LIN {X 0,Y 368.317,Z 1145.734,A -85,B 0,C 180,E1 7410.615,E2 7410.615} C_VEL
LIN {X 0,Y 379.738,Z 1127.366,A -85,B 0,C 180,E1 7408.419,E2 7408.419} C_VEL
LIN {X 0,Y 392.747,Z 1104.648,A -85,B 0,C 180,E1 7406.175,E2 7406.175} C_VEL
LIN {X 0,Y 402.957,Z 1085.189,A -85,B 0,C 180,E1 7404.57,E2 7404.57} C_VEL
LIN {X 0,Y 412.037,Z 1066.456,A -85,B 0,C 180,E1 7403.257,E2 7403.257} C_VEL
LIN {X 0,Y 421.125,Z 1045.858,A -85,B 0,C 180,E1 7402.016,E2 7402.016} C_VEL
LIN {X 0,Y 431.363,Z 1019.668,A -85,B 0,C 180,E1 7400.719,E2 7400.719} C_VEL
LIN {X 0,Y 438.943,Z 997.212,A -85,B 0,C 180,E1 7399.812,E2 7399.812} C_VEL
LIN {X 0,Y 444.979,Z 976.797,A -85,B 0,C 180,E1 7399.128,E2 7399.128} C_VEL
LIN {X 0,Y 450.336,Z 955.699,A -85,B 0,C 180,E1 7398.541,E2 7398.541} C_VEL
LIN {X 0,Y 455.391,Z 931.712,A -85,B 0,C 180,E1 7398.007,E2 7398.007} C_VEL
LIN {X 0,Y 459.835,Z 902.521,A -85,B 0,C 180,E1 7397.489,E2 7397.489} C_VEL
LIN {X 0,Y 466.482,Z 832.802,A -85,B 0,C 180,E1 7396.426,E2 7396.426} C_VEL
LIN {X 0,Y 482.162,Z 665.13,A -85,B 0,C 180,E1 7393.919,E2 7393.919} C_VEL
LIN {X 0,Y 478.75,Z 659.044,A -85,B 0,C 180,E1 7391.75,E2 7391.75} C_VEL
LIN {X 0,Y 476.474,Z 654.994,A -85,B 0,C 180,E1 7390.031,E2 7390.031} C_VEL
LIN {X 0,Y 474.855,Z 652.158,A -85,B 0,C 180,E1 7388.598,E2 7388.598} C_VEL
LIN {X 0,Y 472.633,Z 648.091,A -85,B 0,C 180,E1 7386.072,E2 7386.072} C_VEL
LIN {X 0,Y 470.733,Z 644.319,A -85,B 0,C 180,E1 7382.191,E2 7382.191} C_VEL
LIN {X 0,Y 470.599,Z 643.362,A -85,B 0,C 180,E1 7381.217,E2 7381.217} C_VEL
LIN {X 0,Y 470.644,Z 643.488,A -85,B 0,C 180,E1 7378.296,E2 7378.296} C_VEL
LIN {X 0,Y 472.388,Z 647.837,A -85,B 0,C 180,E1 7374.047,E2 7374.047} C_VEL
LIN {X 0,Y 473.08,Z 648.922,A -85,B 0,C 180,E1 7373.141,E2 7373.141} C_VEL
LIN {X 0,Y 475.759,Z 653.672,A -85,B 0,C 180,E1 7370.382,E2 7370.382} C_VEL
LIN {X 0,Y 478.483,Z 658.51,A -85,B 0,C 180,E1 7368.244,E2 7368.244} C_VEL
LIN {X 0,Y 481.951,Z 664.628,A -85,B 0,C 180,E1 7366.013,E2 7366.013} C_VEL
LIN {X 0,Y 482.096,Z 665.255,A -85,B 0,C 180,E1 7365.906,E2 7365.906} C_VEL
LIN {X 0,Y 461.587,Z 885.46,A -85,B 0,C 180,E1 7362.619,E2 7362.619} C_VEL
LIN {X 0,Y 458.167,Z 912.997,A -85,B 0,C 180,E1 7362.164,E2 7362.164} C_VEL
LIN {X 0,Y 454.312,Z 935.058,A -85,B 0,C 180,E1 7361.738,E2 7361.738} C_VEL
LIN {X 0,Y 449.575,Z 956.787,A -85,B 0,C 180,E1 7361.215,E2 7361.215} C_VEL
LIN {X 0,Y 442.785,Z 982.701,A -85,B 0,C 180,E1 7360.432,E2 7360.432} C_VEL
LIN {X 0,Y 434.59,Z 1008.147,A -85,B 0,C 180,E1 7359.461,E2 7359.461} C_VEL
LIN {X 0,Y 427.121,Z 1028.517,A -85,B 0,C 180,E1 7358.524,E2 7358.524} C_VEL
LIN {X 0,Y 418.998,Z 1048.357,A -85,B 0,C 180,E1 7357.451,E2 7357.451} C_VEL
LIN {X 0,Y 409.164,Z 1070.092,A -85,B 0,C 180,E1 7356.062,E2 7356.062} C_VEL
LIN {X 0,Y 397.169,Z 1093.722,A -85,B 0,C 180,E1 7354.235,E2 7354.235} C_VEL
LIN {X 0,Y 387.044,Z 1111.972,A -85,B 0,C 180,E1 7352.552,E2 7352.552} C_VEL
LIN {X 0,Y 377.466,Z 1128.083,A -85,B 0,C 180,E1 7350.83,E2 7350.83} C_VEL
LIN {X 0,Y 367.103,Z 1144.491,A -85,B 0,C 180,E1 7348.791,E2 7348.791} C_VEL
LIN {X 0,Y 354.544,Z 1163.366,A -85,B 0,C 180,E1 7346.015,E2 7346.015} C_VEL
LIN {X 0,Y 342.233,Z 1180.606,A -85,B 0,C 180,E1 7342.907,E2 7342.907} C_VEL
LIN {X 0,Y 332.469,Z 1193.855,A -85,B 0,C 180,E1 7340.081,E2 7340.081} C_VEL
LIN {X 0,Y 323.49,Z 1205.781,A -85,B 0,C 180,E1 7337.105,E2 7337.105} C_VEL
LIN {X 0,Y 314.469,Z 1217.64,A -85,B 0,C 180,E1 7333.633,E2 7333.633} C_VEL
LIN {X 0,Y 304.257,Z 1231.131,A -85,B 0,C 180,E1 7328.843,E2 7328.843} C_VEL
LIN {X 0,Y 296.916,Z 1241.098,A -85,B 0,C 180,E1 7324.459,E2 7324.459} C_VEL
LIN {X 0,Y 291.438,Z 1249.004,A -85,B 0,C 180,E1 7320.292,E2 7320.292} C_VEL
LIN {X 0,Y 286.992,Z 1256.043,A -85,B 0,C 180,E1 7315.822,E2 7315.822} C_VEL
LIN {X 0,Y 283.199,Z 1263.061,A -85,B 0,C 180,E1 7310.249,E2 7310.249} C_VEL
LIN {X 0,Y 281.158,Z 1267.846,A -85,B 0,C 180,E1 7305.052,E2 7305.052} C_VEL
LIN {X 0,Y 280.319,Z 1270.683,A -85,B 0,C 180,E1 7300.903,E2 7300.903} C_VEL
LIN {X 0,Y 280.001,Z 1272.679,A -85,B 0,C 180,E1 7296.567,E2 7296.567} C_VEL
LIN {X 0,Y 279.918,Z 1273.647,A -85,B 0,C 180,E1 7292.667,E2 7292.667} C_VEL
LIN {X 0,Y 279.893,Z 1273.817,A -85,B 0,C 180,E1 7288.778,E2 7288.778} C_VEL
LIN {X 0,Y 279.952,Z 1273.12,A -85,B 0,C 180,E1 7284.678,E2 7284.678} C_VEL
LIN {X 0,Y 280.164,Z 1271.42,A -85,B 0,C 180,E1 7280.35,E2 7280.35} C_VEL
LIN {X 0,Y 280.87,Z 1268.724,A -85,B 0,C 180,E1 7275.998,E2 7275.998} C_VEL
LIN {X 0,Y 282.28,Z 1265.011,A -85,B 0,C 180,E1 7271.631,E2 7271.631} C_VEL
LIN {X 0,Y 284.588,Z 1260.252,A -85,B 0,C 180,E1 7267.272,E2 7267.272} C_VEL
LIN {X 0,Y 287.983,Z 1254.413,A -85,B 0,C 180,E1 7262.953,E2 7262.953} C_VEL
LIN {X 0,Y 293.535,Z 1246.053,A -85,B 0,C 180,E1 7257.909,E2 7257.909} C_VEL
LIN {X 0,Y 301.122,Z 1235.389,A -85,B 0,C 180,E1 7252.828,E2 7252.828} C_VEL
LIN {X 0,Y 308.625,Z 1225.359,A -85,B 0,C 180,E1 7248.886,E2 7248.886} C_VEL
LIN {X 0,Y 316.874,Z 1214.522,A -85,B 0,C 180,E1 7245.288,E2 7245.288} C_VEL
LIN {X 0,Y 327.702,Z 1200.432,A -85,B 0,C 180,E1 7241.368,E2 7241.368} C_VEL
LIN {X 0,Y 339.429,Z 1184.587,A -85,B 0,C 180,E1 7237.787,E2 7237.787} C_VEL
LIN {X 0,Y 349.631,Z 1170.387,A -85,B 0,C 180,E1 7235.088,E2 7235.088} C_VEL
LIN {X 0,Y 359.883,Z 1155.548,A -85,B 0,C 180,E1 7232.677,E2 7232.677} C_VEL
LIN {X 0,Y 371.153,Z 1138.435,A -85,B 0,C 180,E1 7230.31,E2 7230.31} C_VEL
LIN {X 0,Y 384.378,Z 1116.814,A -85,B 0,C 180,E1 7227.831,E2 7227.831} C_VEL
LIN {X 0,Y 394.621,Z 1098.654,A -85,B 0,C 180,E1 7226.089,E2 7226.089} C_VEL
LIN {X 0,Y 404.103,Z 1080.565,A -85,B 0,C 180,E1 7224.604,E2 7224.604} C_VEL
LIN {X 0,Y 412.057,Z 1064.18,A -85,B 0,C 180,E1 7223.441,E2 7223.441} C_VEL
LIN {X 0,Y 414.616,Z 1057.936,A -85,B 0,C 180,E1 7222.906,E2 7222.906} C_VEL
LIN {X 0,Y 419.105,Z 1042.697,A -85,B 0,C 180,E1 7221.208,E2 7221.208} C_VEL
LIN {X 0,Y 421.394,Z 1036.166,A -85,B 0,C 180,E1 7220.733,E2 7220.733} C_VEL
LIN {X 0,Y 430.003,Z 1013.794,A -85,B 0,C 180,E1 7219.672,E2 7219.672} C_VEL
LIN {X 0,Y 436.87,Z 993.636,A -85,B 0,C 180,E1 7218.864,E2 7218.864} C_VEL
LIN {X 0,Y 443.002,Z 973.077,A -85,B 0,C 180,E1 7218.173,E2 7218.173} C_VEL
LIN {X 0,Y 448.601,Z 951.126,A -85,B 0,C 180,E1 7217.565,E2 7217.565} C_VEL
LIN {X 0,Y 454.241,Z 923.875,A -85,B 0,C 180,E1 7216.969,E2 7216.969} C_VEL
LIN {X 0,Y 458.06,Z 897.621,A -85,B 0,C 180,E1 7216.52,E2 7216.52} C_VEL
LIN {X 0,Y 474.049,Z 730.963,A -85,B 0,C 180,E1 7214.035,E2 7214.035} C_VEL
LIN {X 0,Y 479.819,Z 670.911,A -85,B 0,C 180,E1 7213.129,E2 7213.129} C_VEL
LIN {X 0,Y 476.073,Z 663.972,A -85,B 0,C 180,E1 7210.467,E2 7210.467} C_VEL
LIN {X 0,Y 473.843,Z 660.068,A -85,B 0,C 180,E1 7208.494,E2 7208.494} C_VEL
LIN {X 0,Y 471.708,Z 656.065,A -85,B 0,C 180,E1 7205.962,E2 7205.962} C_VEL
LIN {X 0,Y 469.919,Z 652.326,A -85,B 0,C 180,E1 7201.951,E2 7201.951} C_VEL
LIN {X 0,Y 469.825,Z 651.372,A -85,B 0,C 180,E1 7200.854,E2 7200.854} C_VEL
LIN {X 0,Y 469.866,Z 651.609,A -85,B 0,C 180,E1 7198.781,E2 7198.781} C_VEL
LIN {X 0,Y 471.112,Z 655.393,A -85,B 0,C 180,E1 7195.008,E2 7195.008} C_VEL
LIN {X 0,Y 472.091,Z 656.797,A -85,B 0,C 180,E1 7193.616,E2 7193.616} C_VEL
LIN {X 0,Y 474.785,Z 661.714,A -85,B 0,C 180,E1 7190.729,E2 7190.729} C_VEL
LIN {X 0,Y 477.278,Z 666.333,A -85,B 0,C 180,E1 7188.704,E2 7188.704} C_VEL
LIN {X 0,Y 479.903,Z 671.155,A -85,B 0,C 180,E1 7186.921,E2 7186.921} C_VEL
LIN {X 0,Y 459.204,Z 888.928,A -85,B 0,C 180,E1 7183.693,E2 7183.693} C_VEL
LIN {X 0,Y 455.746,Z 916.161,A -85,B 0,C 180,E1 7183.247,E2 7183.247} C_VEL
LIN {X 0,Y 451.785,Z 938.355,A -85,B 0,C 180,E1 7182.831,E2 7182.831} C_VEL
LIN {X 0,Y 446.979,Z 959.904,A -85,B 0,C 180,E1 7182.335,E2 7182.335} C_VEL
LIN {X 0,Y 440.355,Z 984.664,A -85,B 0,C 180,E1 7181.626,E2 7181.626} C_VEL
LIN {X 0,Y 431.937,Z 1010.547,A -85,B 0,C 180,E1 7180.684,E2 7180.684} C_VEL
LIN {X 0,Y 424.106,Z 1031.526,A -85,B 0,C 180,E1 7179.756,E2 7179.756} C_VEL
LIN {X 0,Y 416.174,Z 1050.594,A -85,B 0,C 180,E1 7178.762,E2 7178.762} C_VEL
LIN {X 0,Y 407.238,Z 1070.13,A -85,B 0,C 180,E1 7177.563,E2 7177.563} C_VEL
LIN {X 0,Y 395.845,Z 1092.788,A -85,B 0,C 180,E1 7175.926,E2 7175.926} C_VEL
LIN {X 0,Y 383.686,Z 1114.369,A -85,B 0,C 180,E1 7174.021,E2 7174.021} C_VEL
LIN {X 0,Y 373.027,Z 1131.965,A -85,B 0,C 180,E1 7172.182,E2 7172.182} C_VEL
LIN {X 0,Y 362.443,Z 1148.392,A -85,B 0,C 180,E1 7170.17,E2 7170.17} C_VEL
LIN {X 0,Y 349.788,Z 1166.999,A -85,B 0,C 180,E1 7167.475,E2 7167.475} C_VEL
LIN {X 0,Y 337.022,Z 1184.513,A -85,B 0,C 180,E1 7164.369,E2 7164.369} C_VEL
LIN {X 0,Y 326.887,Z 1197.959,A -85,B 0,C 180,E1 7161.53,E2 7161.53} C_VEL
LIN {X 0,Y 317.538,Z 1210.075,A -85,B 0,C 180,E1 7158.53,E2 7158.53} C_VEL
LIN {X 0,Y 308.117,Z 1222.135,A -85,B 0,C 180,E1 7155.017,E2 7155.017} C_VEL
LIN {X 0,Y 297.906,Z 1235.366,A -85,B 0,C 180,E1 7150.365,E2 7150.365} C_VEL
LIN {X 0,Y 289.742,Z 1246.09,A -85,B 0,C 180,E1 7145.668,E2 7145.668} C_VEL
LIN {X 0,Y 283.977,Z 1254.183,A -85,B 0,C 180,E1 7141.398,E2 7141.398} C_VEL
LIN {X 0,Y 279.444,Z 1261.114,A -85,B 0,C 180,E1 7137.006,E2 7137.006} C_VEL
LIN {X 0,Y 275.889,Z 1267.394,A -85,B 0,C 180,E1 7132.136,E2 7132.136} C_VEL
LIN {X 0,Y 273.308,Z 1273.104,A -85,B 0,C 180,E1 7126.355,E2 7126.355} C_VEL
LIN {X 0,Y 272.278,Z 1276.597,A -85,B 0,C 180,E1 7121.33,E2 7121.33} C_VEL
LIN {X 0,Y 271.97,Z 1278.637,A -85,B 0,C 180,E1 7116.949,E2 7116.949} C_VEL
LIN {X 0,Y 271.913,Z 1279.663,A -85,B 0,C 180,E1 7112.945,E2 7112.945} C_VEL
LIN {X 0,Y 271.897,Z 1279.844,A -85,B 0,C 180,E1 7108.73,E2 7108.73} C_VEL
LIN {X 0,Y 271.931,Z 1279.107,A -85,B 0,C 180,E1 7104.508,E2 7104.508} C_VEL
LIN {X 0,Y 272.089,Z 1277.448,A -85,B 0,C 180,E1 7100.262,E2 7100.262} C_VEL
LIN {X 0,Y 272.771,Z 1274.701,A -85,B 0,C 180,E1 7095.777,E2 7095.777} C_VEL
LIN {X 0,Y 274.181,Z 1270.916,A -85,B 0,C 180,E1 7091.276,E2 7091.276} C_VEL
LIN {X 0,Y 276.532,Z 1266.069,A -85,B 0,C 180,E1 7086.783,E2 7086.783} C_VEL
LIN {X 0,Y 279.837,Z 1260.434,A -85,B 0,C 180,E1 7082.548,E2 7082.548} C_VEL
LIN {X 0,Y 284.734,Z 1253.054,A -85,B 0,C 180,E1 7077.972,E2 7077.972} C_VEL
LIN {X 0,Y 292.301,Z 1242.694,A -85,B 0,C 180,E1 7072.732,E2 7072.732} C_VEL
LIN {X 0,Y 301.068,Z 1231.11,A -85,B 0,C 180,E1 7068.068,E2 7068.068} C_VEL
LIN {X 0,Y 309.48,Z 1220.307,A -85,B 0,C 180,E1 7064.432,E2 7064.432} C_VEL
LIN {X 0,Y 319.243,Z 1207.822,A -85,B 0,C 180,E1 7060.89,E2 7060.89} C_VEL
LIN {X 0,Y 331.907,Z 1191.336,A -85,B 0,C 180,E1 7057.025,E2 7057.025} C_VEL
LIN {X 0,Y 343.634,Z 1175.359,A -85,B 0,C 180,E1 7053.964,E2 7053.964} C_VEL
LIN {X 0,Y 353.856,Z 1160.909,A -85,B 0,C 180,E1 7051.618,E2 7051.618} C_VEL
LIN {X 0,Y 364.151,Z 1145.639,A -85,B 0,C 180,E1 7049.488,E2 7049.488} C_VEL
LIN {X 0,Y 375.653,Z 1127.607,A -85,B 0,C 180,E1 7047.345,E2 7047.345} C_VEL
LIN {X 0,Y 389.207,Z 1104.505,A -85,B 0,C 180,E1 7045.081,E2 7045.081} C_VEL
LIN {X 0,Y 399.609,Z 1085.094,A -85,B 0,C 180,E1 7043.498,E2 7043.498} C_VEL
LIN {X 0,Y 408.802,Z 1066.504,A -85,B 0,C 180,E1 7042.211,E2 7042.211} C_VEL
LIN {X 0,Y 417.778,Z 1046.575,A -85,B 0,C 180,E1 7041.024,E2 7041.024} C_VEL
LIN {X 0,Y 428.155,Z 1020.705,A -85,B 0,C 180,E1 7039.752,E2 7039.752} C_VEL
LIN {X 0,Y 436.117,Z 997.583,A -85,B 0,C 180,E1 7038.828,E2 7038.828} C_VEL
LIN {X 0,Y 442.334,Z 976.931,A -85,B 0,C 180,E1 7038.147,E2 7038.147} C_VEL
LIN {X 0,Y 447.76,Z 955.926,A -85,B 0,C 180,E1 7037.572,E2 7037.572} C_VEL
LIN {X 0,Y 452.756,Z 932.675,A -85,B 0,C 180,E1 7037.061,E2 7037.061} C_VEL
LIN {X 0,Y 457.442,Z 902.766,A -85,B 0,C 180,E1 7036.534,E2 7036.534} C_VEL
LIN {X 0,Y 463.818,Z 837.541,A -85,B 0,C 180,E1 7035.546,E2 7035.546} C_VEL
LIN {X 0,Y 479.71,Z 670.904,A -85,B 0,C 180,E1 7033.071,E2 7033.071} C_VEL
LIN {X 0,Y 475.936,Z 663.895,A -85,B 0,C 180,E1 7030.409,E2 7030.409} C_VEL
LIN {X 0,Y 473.747,Z 660.045,A -85,B 0,C 180,E1 7028.496,E2 7028.496} C_VEL
LIN {X 0,Y 471.564,Z 655.972,A -85,B 0,C 180,E1 7025.964,E2 7025.964} C_VEL
LIN {X 0,Y 469.727,Z 652.2,A -85,B 0,C 180,E1 7022.074,E2 7022.074} C_VEL
LIN {X 0,Y 469.602,Z 651.303,A -85,B 0,C 180,E1 7021.098,E2 7021.098} C_VEL
LIN {X 0,Y 469.657,Z 651.529,A -85,B 0,C 180,E1 7018.292,E2 7018.292} C_VEL
LIN {X 0,Y 471.506,Z 655.906,A -85,B 0,C 180,E1 7013.913,E2 7013.913} C_VEL
LIN {X 0,Y 474.501,Z 661.361,A -85,B 0,C 180,E1 7010.601,E2 7010.601} C_VEL
LIN {X 0,Y 477.157,Z 666.206,A -85,B 0,C 180,E1 7008.456,E2 7008.456} C_VEL
LIN {X 0,Y 479.675,Z 670.8,A -85,B 0,C 180,E1 7006.755,E2 7006.755} C_VEL
LIN {X 0,Y 458.737,Z 890.156,A -85,B 0,C 180,E1 7003.501,E2 7003.501} C_VEL
LIN {X 0,Y 455.594,Z 914.237,A -85,B 0,C 180,E1 7003.104,E2 7003.104} C_VEL
LIN {X 0,Y 451.679,Z 936.071,A -85,B 0,C 180,E1 7002.685,E2 7002.685} C_VEL
LIN {X 0,Y 446.64,Z 958.608,A -85,B 0,C 180,E1 7002.146,E2 7002.146} C_VEL
LIN {X 0,Y 438.862,Z 986.854,A -85,B 0,C 180,E1 7001.281,E2 7001.281} C_VEL
LIN {X 0,Y 431.414,Z 1009.371,A -85,B 0,C 180,E1 7000.419,E2 7000.419} C_VEL
LIN {X 0,Y 423.82,Z 1029.615,A -85,B 0,C 180,E1 6999.494,E2 6999.494} C_VEL
LIN {X 0,Y 415.522,Z 1049.426,A -85,B 0,C 180,E1 6998.431,E2 6998.431} C_VEL
LIN {X 0,Y 404.396,Z 1073.352,A -85,B 0,C 180,E1 6996.899,E2 6996.899} C_VEL
LIN {X 0,Y 393.143,Z 1094.765,A -85,B 0,C 180,E1 6995.23,E2 6995.23} C_VEL
LIN {X 0,Y 383.352,Z 1112.005,A -85,B 0,C 180,E1 6993.651,E2 6993.651} C_VEL
LIN {X 0,Y 373.422,Z 1128.307,A -85,B 0,C 180,E1 6991.923,E2 6991.923} C_VEL
LIN {X 0,Y 362.775,Z 1144.736,A -85,B 0,C 180,E1 6989.892,E2 6989.892} C_VEL
LIN {X 0,Y 349.751,Z 1163.743,A -85,B 0,C 180,E1 6987.099,E2 6987.099} C_VEL
LIN {X 0,Y 337.257,Z 1180.7,A -85,B 0,C 180,E1 6984.04,E2 6984.04} C_VEL
LIN {X 0,Y 327.152,Z 1193.959,A -85,B 0,C 180,E1 6981.204,E2 6981.204} C_VEL
LIN {X 0,Y 317.349,Z 1206.506,A -85,B 0,C 180,E1 6978.042,E2 6978.042} C_VEL
LIN {X 0,Y 306.719,Z 1220.011,A -85,B 0,C 180,E1 6973.982,E2 6973.982} C_VEL
LIN {X 0,Y 296.734,Z 1232.51,A -85,B 0,C 180,E1 6969.313,E2 6969.313} C_VEL
LIN {X 0,Y 289.758,Z 1241.592,A -85,B 0,C 180,E1 6965.194,E2 6965.194} C_VEL
LIN {X 0,Y 284.027,Z 1249.446,A -85,B 0,C 180,E1 6960.934,E2 6960.934} C_VEL
LIN {X 0,Y 278.966,Z 1257.098,A -85,B 0,C 180,E1 6955.887,E2 6955.887} C_VEL
LIN {X 0,Y 275.042,Z 1263.966,A -85,B 0,C 180,E1 6949.988,E2 6949.988} C_VEL
LIN {X 0,Y 273.214,Z 1268.093,A -85,B 0,C 180,E1 6945.283,E2 6945.283} C_VEL
LIN {X 0,Y 272.335,Z 1270.884,A -85,B 0,C 180,E1 6941.012,E2 6941.012} C_VEL
LIN {X 0,Y 272.008,Z 1272.767,A -85,B 0,C 180,E1 6936.761,E2 6936.761} C_VEL
LIN {X 0,Y 271.919,Z 1273.735,A -85,B 0,C 180,E1 6932.746,E2 6932.746} C_VEL
LIN {X 0,Y 271.896,Z 1273.904,A -85,B 0,C 180,E1 6928.742,E2 6928.742} C_VEL
LIN {X 0,Y 271.957,Z 1273.208,A -85,B 0,C 180,E1 6924.521,E2 6924.521} C_VEL
LIN {X 0,Y 272.186,Z 1271.508,A -85,B 0,C 180,E1 6920.064,E2 6920.064} C_VEL
LIN {X 0,Y 272.968,Z 1268.813,A -85,B 0,C 180,E1 6915.584,E2 6915.584} C_VEL
LIN {X 0,Y 274.49,Z 1265.1,A -85,B 0,C 180,E1 6911.09,E2 6911.09} C_VEL
LIN {X 0,Y 276.97,Z 1260.341,A -85,B 0,C 180,E1 6906.61,E2 6906.61} C_VEL
LIN {X 0,Y 280.597,Z 1254.503,A -85,B 0,C 180,E1 6902.181,E2 6902.181} C_VEL
LIN {X 0,Y 286.485,Z 1246.143,A -85,B 0,C 180,E1 6897.02,E2 6897.02} C_VEL
LIN {X 0,Y 294.492,Z 1235.479,A -85,B 0,C 180,E1 6891.843,E2 6891.843} C_VEL
LIN {X 0,Y 302.347,Z 1225.449,A -85,B 0,C 180,E1 6887.839,E2 6887.839} C_VEL
LIN {X 0,Y 310.97,Z 1214.612,A -85,B 0,C 180,E1 6884.2,E2 6884.2} C_VEL
LIN {X 0,Y 322.229,Z 1200.522,A -85,B 0,C 180,E1 6880.251,E2 6880.251} C_VEL
LIN {X 0,Y 334.193,Z 1184.921,A -85,B 0,C 180,E1 6876.706,E2 6876.706} C_VEL
LIN {X 0,Y 344.807,Z 1170.617,A -85,B 0,C 180,E1 6873.98,E2 6873.98} C_VEL
LIN {X 0,Y 355.468,Z 1155.636,A -85,B 0,C 180,E1 6871.55,E2 6871.55} C_VEL
LIN {X 0,Y 367.136,Z 1138.387,A -85,B 0,C 180,E1 6869.177,E2 6869.177} C_VEL
LIN {X 0,Y 380.601,Z 1116.9,A -85,B 0,C 180,E1 6866.734,E2 6866.734} C_VEL
LIN {X 0,Y 391.078,Z 1098.74,A -85,B 0,C 180,E1 6865.008,E2 6865.008} C_VEL
LIN {X 0,Y 400.88,Z 1080.414,A -85,B 0,C 180,E1 6863.521,E2 6863.521} C_VEL
LIN {X 0,Y 409.928,Z 1062.06,A -85,B 0,C 180,E1 6862.248,E2 6862.248} C_VEL
LIN {X 0,Y 420.216,Z 1039.054,A -85,B 0,C 180,E1 6860.884,E2 6860.884} C_VEL
LIN {X 0,Y 421.394,Z 1036.166,A -85,B 0,C 180,E1 6860.733,E2 6860.733} C_VEL
LIN {X 0,Y 423.713,Z 1029.54,A -85,B 0,C 180,E1 6860.279,E2 6860.279} C_VEL
LIN {X 0,Y 428.122,Z 1012.463,A -85,B 0,C 180,E1 6858.69,E2 6858.69} C_VEL
LIN {X 0,Y 429.972,Z 1006.631,A -85,B 0,C 180,E1 6858.346,E2 6858.346} C_VEL
LIN {X 0,Y 438.893,Z 979.066,A -85,B 0,C 180,E1 6857.359,E2 6857.359} C_VEL
LIN {X 0,Y 445.082,Z 955.962,A -85,B 0,C 180,E1 6856.699,E2 6856.699} C_VEL
LIN {X 0,Y 449.846,Z 934.642,A -85,B 0,C 180,E1 6856.209,E2 6856.209} C_VEL
LIN {X 0,Y 453.871,Z 912.105,A -85,B 0,C 180,E1 6855.79,E2 6855.79} C_VEL
LIN {X 0,Y 457.572,Z 882.153,A -85,B 0,C 180,E1 6855.312,E2 6855.312} C_VEL
LIN {X 0,Y 477.509,Z 676.816,A -85,B 0,C 180,E1 6852.294,E2 6852.294} C_VEL
LIN {X 0,Y 474.281,Z 670.822,A -85,B 0,C 180,E1 6849.832,E2 6849.832} C_VEL
LIN {X 0,Y 472.616,Z 667.782,A -85,B 0,C 180,E1 6848.272,E2 6848.272} C_VEL
LIN {X 0,Y 470.643,Z 663.947,A -85,B 0,C 180,E1 6845.853,E2 6845.853} C_VEL
LIN {X 0,Y 468.92,Z 660.205,A -85,B 0,C 180,E1 6841.833,E2 6841.833} C_VEL
LIN {X 0,Y 468.836,Z 659.318,A -85,B 0,C 180,E1 6840.733,E2 6840.733} C_VEL
LIN {X 0,Y 468.883,Z 659.62,A -85,B 0,C 180,E1 6838.778,E2 6838.778} C_VEL
LIN {X 0,Y 470.135,Z 663.376,A -85,B 0,C 180,E1 6834.997,E2 6834.997} C_VEL
LIN {X 0,Y 471.013,Z 664.714,A -85,B 0,C 180,E1 6833.723,E2 6833.723} C_VEL
LIN {X 0,Y 473.596,Z 669.536,A -85,B 0,C 180,E1 6830.889,E2 6830.889} C_VEL
LIN {X 0,Y 476.04,Z 674.176,A -85,B 0,C 180,E1 6828.858,E2 6828.858} C_VEL
LIN {X 0,Y 477.549,Z 677.122,A -85,B 0,C 180,E1 6827.772,E2 6827.772} C_VEL
LIN {X 0,Y 456.473,Z 893.486,A -85,B 0,C 180,E1 6824.588,E2 6824.588} C_VEL
LIN {X 0,Y 453.312,Z 917.226,A -85,B 0,C 180,E1 6824.199,E2 6824.199} C_VEL
LIN {X 0,Y 449.265,Z 939.323,A -85,B 0,C 180,E1 6823.789,E2 6823.789} C_VEL
LIN {X 0,Y 443.992,Z 962.337,A -85,B 0,C 180,E1 6823.262,E2 6823.262} C_VEL
LIN {X 0,Y 435.92,Z 990.787,A -85,B 0,C 180,E1 6822.424,E2 6822.424} C_VEL
LIN {X 0,Y 428.73,Z 1012.087,A -85,B 0,C 180,E1 6821.64,E2 6821.64} C_VEL
LIN {X 0,Y 421.359,Z 1031.443,A -85,B 0,C 180,E1 6820.794,E2 6820.794} C_VEL
LIN {X 0,Y 413.287,Z 1050.51,A -85,B 0,C 180,E1 6819.817,E2 6819.817} C_VEL
LIN {X 0,Y 404.181,Z 1070.046,A -85,B 0,C 180,E1 6818.637,E2 6818.637} C_VEL
LIN {X 0,Y 392.174,Z 1093.382,A -85,B 0,C 180,E1 6816.968,E2 6816.968} C_VEL
LIN {X 0,Y 380.134,Z 1114.282,A -85,B 0,C 180,E1 6815.142,E2 6815.142} C_VEL
LIN {X 0,Y 369.228,Z 1131.878,A -85,B 0,C 180,E1 6813.321,E2 6813.321} C_VEL
LIN {X 0,Y 358.363,Z 1148.327,A -85,B 0,C 180,E1 6811.321,E2 6811.321} C_VEL
LIN {X 0,Y 345.37,Z 1166.911,A -85,B 0,C 180,E1 6808.642,E2 6808.642} C_VEL
LIN {X 0,Y 332.163,Z 1184.48,A -85,B 0,C 180,E1 6805.533,E2 6805.533} C_VEL
LIN {X 0,Y 321.703,Z 1197.903,A -85,B 0,C 180,E1 6802.693,E2 6802.693} C_VEL
LIN {X 0,Y 311.514,Z 1210.624,A -85,B 0,C 180,E1 6799.516,E2 6799.516} C_VEL
LIN {X 0,Y 300.85,Z 1223.776,A -85,B 0,C 180,E1 6795.597,E2 6795.597} C_VEL
LIN {X 0,Y 289.982,Z 1237.126,A -85,B 0,C 180,E1 6790.659,E2 6790.659} C_VEL
LIN {X 0,Y 282.636,Z 1246.408,A -85,B 0,C 180,E1 6786.456,E2 6786.456} C_VEL
LIN {X 0,Y 276.605,Z 1254.449,A -85,B 0,C 180,E1 6782.09,E2 6782.09} C_VEL
LIN {X 0,Y 271.665,Z 1261.617,A -85,B 0,C 180,E1 6777.384,E2 6777.384} C_VEL
LIN {X 0,Y 267.419,Z 1268.839,A -85,B 0,C 180,E1 6771.405,E2 6771.405} C_VEL
LIN {X 0,Y 265.244,Z 1273.501,A -85,B 0,C 180,E1 6766.191,E2 6766.191} C_VEL
LIN {X 0,Y 264.302,Z 1276.588,A -85,B 0,C 180,E1 6761.525,E2 6761.525} C_VEL
LIN {X 0,Y 263.973,Z 1278.582,A -85,B 0,C 180,E1 6757.058,E2 6757.058} C_VEL
LIN {X 0,Y 263.913,Z 1279.599,A -85,B 0,C 180,E1 6752.817,E2 6752.817} C_VEL
LIN {X 0,Y 263.898,Z 1279.757,A -85,B 0,C 180,E1 6748.691,E2 6748.691} C_VEL
LIN {X 0,Y 263.934,Z 1279.019,A -85,B 0,C 180,E1 6744.341,E2 6744.341} C_VEL
LIN {X 0,Y 264.121,Z 1277.289,A -85,B 0,C 180,E1 6739.832,E2 6739.832} C_VEL
LIN {X 0,Y 264.864,Z 1274.611,A -85,B 0,C 180,E1 6735.343,E2 6735.343} C_VEL
LIN {X 0,Y 266.397,Z 1270.825,A -85,B 0,C 180,E1 6730.708,E2 6730.708} C_VEL
LIN {X 0,Y 268.928,Z 1265.977,A -85,B 0,C 180,E1 6726.087,E2 6726.087} C_VEL
LIN {X 0,Y 272.462,Z 1260.337,A -85,B 0,C 180,E1 6721.735,E2 6721.735} C_VEL
LIN {X 0,Y 277.394,Z 1253.318,A -85,B 0,C 180,E1 6717.264,E2 6717.264} C_VEL
LIN {X 0,Y 285.315,Z 1243.059,A -85,B 0,C 180,E1 6711.912,E2 6711.912} C_VEL
LIN {X 0,Y 294.372,Z 1231.621,A -85,B 0,C 180,E1 6707.196,E2 6707.196} C_VEL
LIN {X 0,Y 303.176,Z 1220.791,A -85,B 0,C 180,E1 6703.479,E2 6703.479} C_VEL
LIN {X 0,Y 312.571,Z 1209.229,A -85,B 0,C 180,E1 6700.129,E2 6700.129} C_VEL
LIN {X 0,Y 324.028,Z 1194.914,A -85,B 0,C 180,E1 6696.644,E2 6696.644} C_VEL
LIN {X 0,Y 337.765,Z 1176.982,A -85,B 0,C 180,E1 6693.09,E2 6693.09} C_VEL
LIN {X 0,Y 348.965,Z 1161.64,A -85,B 0,C 180,E1 6690.576,E2 6690.576} C_VEL
LIN {X 0,Y 359.438,Z 1146.563,A -85,B 0,C 180,E1 6688.467,E2 6688.467} C_VEL
LIN {X 0,Y 369.97,Z 1130.522,A -85,B 0,C 180,E1 6686.543,E2 6686.543} C_VEL
LIN {X 0,Y 382.391,Z 1110.344,A -85,B 0,C 180,E1 6684.496,E2 6684.496} C_VEL
LIN {X 0,Y 395.249,Z 1087.21,A -85,B 0,C 180,E1 6682.573,E2 6682.573} C_VEL
LIN {X 0,Y 405.086,Z 1067.834,A -85,B 0,C 180,E1 6681.231,E2 6681.231} C_VEL
LIN {X 0,Y 413.715,Z 1049.187,A -85,B 0,C 180,E1 6680.12,E2 6680.12} C_VEL
LIN {X 0,Y 422.204,Z 1028.957,A -85,B 0,C 180,E1 6679.098,E2 6679.098} C_VEL
LIN {X 0,Y 431.657,Z 1003.454,A -85,B 0,C 180,E1 6678.029,E2 6678.029} C_VEL
LIN {X 0,Y 439.257,Z 979.058,A -85,B 0,C 180,E1 6677.213,E2 6677.213} C_VEL
LIN {X 0,Y 444.945,Z 957.673,A -85,B 0,C 180,E1 6676.629,E2 6676.629} C_VEL
LIN {X 0,Y 449.718,Z 936.208,A -85,B 0,C 180,E1 6676.155,E2 6676.155} C_VEL
LIN {X 0,Y 454.156,Z 910.846,A -85,B 0,C 180,E1 6675.697,E2 6675.697} C_VEL
LIN {X 0,Y 458.264,Z 873.736,A -85,B 0,C 180,E1 6675.122,E2 6675.122} C_VEL
LIN {X 0,Y 477.37,Z 676.767,A -85,B 0,C 180,E1 6672.223,E2 6672.223} C_VEL
LIN {X 0,Y 474.135,Z 670.741,A -85,B 0,C 180,E1 6669.774,E2 6669.774} C_VEL
LIN {X 0,Y 472.392,Z 667.581,A -85,B 0,C 180,E1 6668.153,E2 6668.153} C_VEL
LIN {X 0,Y 470.406,Z 663.755,A -85,B 0,C 180,E1 6665.734,E2 6665.734} C_VEL
LIN {X 0,Y 468.707,Z 659.928,A -85,B 0,C 180,E1 6661.834,E2 6661.834} C_VEL
LIN {X 0,Y 468.607,Z 659.246,A -85,B 0,C 180,E1 6660.978,E2 6660.978} C_VEL
LIN {X 0,Y 468.663,Z 659.411,A -85,B 0,C 180,E1 6658.411,E2 6658.411} C_VEL
LIN {X 0,Y 470.44,Z 663.788,A -85,B 0,C 180,E1 6654.022,E2 6654.022} C_VEL
LIN {X 0,Y 473.25,Z 669.051,A -85,B 0,C 180,E1 6650.821,E2 6650.821} C_VEL
LIN {X 0,Y 475.917,Z 674.051,A -85,B 0,C 180,E1 6648.61,E2 6648.61} C_VEL
LIN {X 0,Y 477.315,Z 676.801,A -85,B 0,C 180,E1 6647.606,E2 6647.606} C_VEL
LIN {X 0,Y 456.2,Z 893.047,A -85,B 0,C 180,E1 6644.423,E2 6644.423} C_VEL
LIN {X 0,Y 453.118,Z 915.639,A -85,B 0,C 180,E1 6644.052,E2 6644.052} C_VEL
LIN {X 0,Y 449.039,Z 937.734,A -85,B 0,C 180,E1 6643.63,E2 6643.63} C_VEL
LIN {X 0,Y 443.064,Z 963.621,A -85,B 0,C 180,E1 6643.003,E2 6643.003} C_VEL
LIN {X 0,Y 435.768,Z 988.708,A -85,B 0,C 180,E1 6642.224,E2 6642.224} C_VEL
LIN {X 0,Y 428.769,Z 1009.467,A -85,B 0,C 180,E1 6641.438,E2 6641.438} C_VEL
LIN {X 0,Y 421.046,Z 1029.71,A -85,B 0,C 180,E1 6640.528,E2 6640.528} C_VEL
LIN {X 0,Y 412.631,Z 1049.445,A -85,B 0,C 180,E1 6639.487,E2 6639.487} C_VEL
LIN {X 0,Y 401.261,Z 1073.446,A -85,B 0,C 180,E1 6637.972,E2 6637.972} C_VEL
LIN {X 0,Y 389.543,Z 1095.274,A -85,B 0,C 180,E1 6636.289,E2 6636.289} C_VEL
LIN {X 0,Y 379.633,Z 1112.322,A -85,B 0,C 180,E1 6634.743,E2 6634.743} C_VEL
LIN {X 0,Y 369.248,Z 1128.954,A -85,B 0,C 180,E1 6632.991,E2 6632.991} C_VEL
LIN {X 0,Y 357.769,Z 1146.193,A -85,B 0,C 180,E1 6630.857,E2 6630.857} C_VEL
LIN {X 0,Y 342.943,Z 1166.925,A -85,B 0,C 180,E1 6627.733,E2 6627.733} C_VEL
LIN {X 0,Y 331.821,Z 1181.56,A -85,B 0,C 180,E1 6625.052,E2 6625.052} C_VEL
LIN {X 0,Y 321.424,Z 1194.739,A -85,B 0,C 180,E1 6622.204,E2 6622.204} C_VEL
LIN {X 0,Y 311.298,Z 1207.231,A -85,B 0,C 180,E1 6619.015,E2 6619.015} C_VEL
LIN {X 0,Y 299.846,Z 1221.193,A -85,B 0,C 180,E1 6614.723,E2 6614.723} C_VEL
LIN {X 0,Y 289.918,Z 1233.058,A -85,B 0,C 180,E1 6610.166,E2 6610.166} C_VEL
LIN {X 0,Y 282.967,Z 1241.685,A -85,B 0,C 180,E1 6606.17,E2 6606.17} C_VEL
LIN {X 0,Y 276.91,Z 1249.538,A -85,B 0,C 180,E1 6601.821,E2 6601.821} C_VEL
LIN {X 0,Y 271.565,Z 1257.126,A -85,B 0,C 180,E1 6596.698,E2 6596.698} C_VEL
LIN {X 0,Y 267.313,Z 1264.057,A -85,B 0,C 180,E1 6590.591,E2 6590.591} C_VEL
LIN {X 0,Y 265.334,Z 1268.183,A -85,B 0,C 180,E1 6585.749,E2 6585.749} C_VEL
LIN {X 0,Y 264.392,Z 1270.973,A -85,B 0,C 180,E1 6581.347,E2 6581.347} C_VEL
LIN {X 0,Y 264.018,Z 1272.855,A -85,B 0,C 180,E1 6576.967,E2 6576.967} C_VEL
LIN {X 0,Y 263.92,Z 1273.823,A -85,B 0,C 180,E1 6572.829,E2 6572.829} C_VEL
LIN {X 0,Y 263.897,Z 1273.992,A -85,B 0,C 180,E1 6568.704,E2 6568.704} C_VEL
LIN {X 0,Y 263.963,Z 1273.296,A -85,B 0,C 180,E1 6564.354,E2 6564.354} C_VEL
LIN {X 0,Y 264.196,Z 1271.708,A -85,B 0,C 180,E1 6559.981,E2 6559.981} C_VEL
LIN {X 0,Y 265.02,Z 1269.059,A -85,B 0,C 180,E1 6555.365,E2 6555.365} C_VEL
LIN {X 0,Y 266.625,Z 1265.393,A -85,B 0,C 180,E1 6550.738,E2 6550.738} C_VEL
LIN {X 0,Y 269.24,Z 1260.682,A -85,B 0,C 180,E1 6546.129,E2 6546.129} C_VEL
LIN {X 0,Y 272.846,Z 1255.192,A -85,B 0,C 180,E1 6541.796,E2 6541.796} C_VEL
LIN {X 0,Y 277.85,Z 1248.331,A -85,B 0,C 180,E1 6537.339,E2 6537.339} C_VEL
LIN {X 0,Y 285.137,Z 1239.09,A -85,B 0,C 180,E1 6532.408,E2 6532.408} C_VEL
LIN {X 0,Y 294.933,Z 1227.071,A -85,B 0,C 180,E1 6527.319,E2 6527.319} C_VEL
LIN {X 0,Y 303.76,Z 1216.409,A -85,B 0,C 180,E1 6523.611,E2 6523.611} C_VEL
LIN {X 0,Y 313.168,Z 1205.027,A -85,B 0,C 180,E1 6520.275,E2 6520.275} C_VEL
LIN {X 0,Y 323.83,Z 1191.874,A -85,B 0,C 180,E1 6517.021,E2 6517.021} C_VEL
LIN {X 0,Y 338.344,Z 1173.228,A -85,B 0,C 180,E1 6513.258,E2 6513.258} C_VEL
LIN {X 0,Y 349.538,Z 1158.028,A -85,B 0,C 180,E1 6510.741,E2 6510.741} C_VEL
LIN {X 0,Y 360.298,Z 1142.647,A -85,B 0,C 180,E1 6508.572,E2 6508.572} C_VEL
LIN {X 0,Y 371.173,Z 1126.171,A -85,B 0,C 180,E1 6506.589,E2 6506.589} C_VEL
LIN {X 0,Y 384.322,Z 1104.814,A -85,B 0,C 180,E1 6504.429,E2 6504.429} C_VEL
LIN {X 0,Y 396.408,Z 1082.932,A -85,B 0,C 180,E1 6502.621,E2 6502.621} C_VEL
LIN {X 0,Y 405.73,Z 1064.572,A -85,B 0,C 180,E1 6501.34,E2 6501.34} C_VEL
LIN {X 0,Y 414.416,Z 1045.784,A -85,B 0,C 180,E1 6500.207,E2 6500.207} C_VEL
LIN {X 0,Y 423.272,Z 1024.609,A -85,B 0,C 180,E1 6499.126,E2 6499.126} C_VEL
LIN {X 0,Y 429.972,Z 1006.631,A -85,B 0,C 180,E1 6498.346,E2 6498.346} C_VEL
LIN {X 0,Y 431.861,Z 1000.737,A -85,B 0,C 180,E1 6498.018,E2 6498.018} C_VEL
LIN {X 0,Y 435.997,Z 981.891,A -85,B 0,C 180,E1 6496.533,E2 6496.533} C_VEL
LIN {X 0,Y 437.508,Z 975.802,A -85,B 0,C 180,E1 6496.247,E2 6496.247} C_VEL
LIN {X 0,Y 443.201,Z 954.569,A -85,B 0,C 180,E1 6495.667,E2 6495.667} C_VEL
LIN {X 0,Y 447.992,Z 933.154,A -85,B 0,C 180,E1 6495.19,E2 6495.19} C_VEL
LIN {X 0,Y 452.63,Z 906.826,A -85,B 0,C 180,E1 6494.719,E2 6494.719} C_VEL
LIN {X 0,Y 456.983,Z 867.132,A -85,B 0,C 180,E1 6494.117,E2 6494.117} C_VEL
LIN {X 0,Y 475.267,Z 682.813,A -85,B 0,C 180,E1 6491.437,E2 6491.437} C_VEL
LIN {X 0,Y 472.682,Z 677.885,A -85,B 0,C 180,E1 6489.313,E2 6489.313} C_VEL
LIN {X 0,Y 471.28,Z 675.317,A -85,B 0,C 180,E1 6487.927,E2 6487.927} C_VEL
LIN {X 0,Y 469.494,Z 671.734,A -85,B 0,C 180,E1 6485.622,E2 6485.622} C_VEL
LIN {X 0,Y 467.913,Z 667.941,A -85,B 0,C 180,E1 6481.592,E2 6481.592} C_VEL
LIN {X 0,Y 467.85,Z 667.263,A -85,B 0,C 180,E1 6480.612,E2 6480.612} C_VEL
LIN {X 0,Y 467.894,Z 667.498,A -85,B 0,C 180,E1 6478.898,E2 6478.898} C_VEL
LIN {X 0,Y 469.084,Z 671.256,A -85,B 0,C 180,E1 6475.109,E2 6475.109} C_VEL
LIN {X 0,Y 469.938,Z 672.63,A -85,B 0,C 180,E1 6473.832,E2 6473.832} C_VEL
LIN {X 0,Y 472.348,Z 677.225,A -85,B 0,C 180,E1 6471.11,E2 6471.11} C_VEL
LIN {X 0,Y 474.884,Z 682.164,A -85,B 0,C 180,E1 6468.954,E2 6468.954} C_VEL
LIN {X 0,Y 475.302,Z 683.085,A -85,B 0,C 180,E1 6468.63,E2 6468.63} C_VEL
LIN {X 0,Y 454.033,Z 896.526,A -85,B 0,C 180,E1 6465.517,E2 6465.517} C_VEL
LIN {X 0,Y 450.924,Z 918.778,A -85,B 0,C 180,E1 6465.153,E2 6465.153} C_VEL
LIN {X 0,Y 446.577,Z 941.726,A -85,B 0,C 180,E1 6464.729,E2 6464.729} C_VEL
LIN {X 0,Y 439.788,Z 969.69,A -85,B 0,C 180,E1 6464.072,E2 6464.072} C_VEL
LIN {X 0,Y 432.982,Z 992.416,A -85,B 0,C 180,E1 6463.385,E2 6463.385} C_VEL
LIN {X 0,Y 425.826,Z 1013.136,A -85,B 0,C 180,E1 6462.63,E2 6462.63} C_VEL
LIN {X 0,Y 417.927,Z 1033.374,A -85,B 0,C 180,E1 6461.751,E2 6461.751} C_VEL
LIN {X 0,Y 408.918,Z 1054.036,A -85,B 0,C 180,E1 6460.688,E2 6460.688} C_VEL
LIN {X 0,Y 396.493,Z 1079.367,A -85,B 0,C 180,E1 6459.103,E2 6459.103} C_VEL
LIN {X 0,Y 385.922,Z 1098.653,A -85,B 0,C 180,E1 6457.643,E2 6457.643} C_VEL
LIN {X 0,Y 375.873,Z 1115.588,A -85,B 0,C 180,E1 6456.15,E2 6456.15} C_VEL
LIN {X 0,Y 364.849,Z 1132.905,A -85,B 0,C 180,E1 6454.359,E2 6454.359} C_VEL
LIN {X 0,Y 352.707,Z 1150.76,A -85,B 0,C 180,E1 6452.173,E2 6452.173} C_VEL
LIN {X 0,Y 337.772,Z 1171.12,A -85,B 0,C 180,E1 6449.131,E2 6449.131} C_VEL
LIN {X 0,Y 326.295,Z 1185.883,A -85,B 0,C 180,E1 6446.448,E2 6446.448} C_VEL
LIN {X 0,Y 315.551,Z 1199.188,A -85,B 0,C 180,E1 6443.583,E2 6443.583} C_VEL
LIN {X 0,Y 304.518,Z 1212.465,A -85,B 0,C 180,E1 6440.187,E2 6440.187} C_VEL
LIN {X 0,Y 291.778,Z 1227.48,A -85,B 0,C 180,E1 6435.452,E2 6435.452} C_VEL
LIN {X 0,Y 282.459,Z 1238.423,A -85,B 0,C 180,E1 6431.17,E2 6431.17} C_VEL
LIN {X 0,Y 275.256,Z 1247.135,A -85,B 0,C 180,E1 6427.076,E2 6427.076} C_VEL
LIN {X 0,Y 268.72,Z 1255.464,A -85,B 0,C 180,E1 6422.365,E2 6422.365} C_VEL
LIN {X 0,Y 262.578,Z 1264.126,A -85,B 0,C 180,E1 6416.206,E2 6416.206} C_VEL
LIN {X 0,Y 259.143,Z 1269.763,A -85,B 0,C 180,E1 6410.973,E2 6410.973} C_VEL
LIN {X 0,Y 257.246,Z 1273.737,A -85,B 0,C 180,E1 6406.244,E2 6406.244} C_VEL
LIN {X 0,Y 256.321,Z 1276.597,A -85,B 0,C 180,E1 6401.696,E2 6401.696} C_VEL
LIN {X 0,Y 255.977,Z 1278.526,A -85,B 0,C 180,E1 6397.174,E2 6397.174} C_VEL
LIN {X 0,Y 255.914,Z 1279.511,A -85,B 0,C 180,E1 6392.905,E2 6392.905} C_VEL
LIN {X 0,Y 255.9,Z 1279.669,A -85,B 0,C 180,E1 6388.65,E2 6388.65} C_VEL
LIN {X 0,Y 255.939,Z 1278.931,A -85,B 0,C 180,E1 6384.164,E2 6384.164} C_VEL
LIN {X 0,Y 256.138,Z 1277.27,A -85,B 0,C 180,E1 6379.649,E2 6379.649} C_VEL
LIN {X 0,Y 256.964,Z 1274.521,A -85,B 0,C 180,E1 6374.882,E2 6374.882} C_VEL
LIN {X 0,Y 258.635,Z 1270.734,A -85,B 0,C 180,E1 6370.105,E2 6370.105} C_VEL
LIN {X 0,Y 261.368,Z 1265.886,A -85,B 0,C 180,E1 6365.35,E2 6365.35} C_VEL
LIN {X 0,Y 265.136,Z 1260.249,A -85,B 0,C 180,E1 6360.884,E2 6360.884} C_VEL
LIN {X 0,Y 270.373,Z 1253.225,A -85,B 0,C 180,E1 6356.303,E2 6356.303} C_VEL
LIN {X 0,Y 278.74,Z 1242.965,A -85,B 0,C 180,E1 6350.845,E2 6350.845} C_VEL
LIN {X 0,Y 288.674,Z 1231.022,A -85,B 0,C 180,E1 6345.871,E2 6345.871} C_VEL
LIN {X 0,Y 297.948,Z 1220.12,A -85,B 0,C 180,E1 6342.122,E2 6342.122} C_VEL
LIN {X 0,Y 308.301,Z 1207.857,A -85,B 0,C 180,E1 6338.586,E2 6338.586} C_VEL
LIN {X 0,Y 321.47,Z 1191.922,A -85,B 0,C 180,E1 6334.796,E2 6334.796} C_VEL
LIN {X 0,Y 334.541,Z 1175.189,A -85,B 0,C 180,E1 6331.585,E2 6331.585} C_VEL
LIN {X 0,Y 345.492,Z 1160.58,A -85,B 0,C 180,E1 6329.236,E2 6329.236} C_VEL
LIN {X 0,Y 356.26,Z 1145.451,A -85,B 0,C 180,E1 6327.159,E2 6327.159} C_VEL
LIN {X 0,Y 367.82,Z 1128.199,A -85,B 0,C 180,E1 6325.14,E2 6325.14} C_VEL
LIN {X 0,Y 382.1,Z 1105.035,A -85,B 0,C 180,E1 6322.905,E2 6322.905} C_VEL
LIN {X 0,Y 392.953,Z 1085.642,A -85,B 0,C 180,E1 6321.356,E2 6321.356} C_VEL
LIN {X 0,Y 402.491,Z 1067.128,A -85,B 0,C 180,E1 6320.103,E2 6320.103} C_VEL
LIN {X 0,Y 411.683,Z 1047.536,A -85,B 0,C 180,E1 6318.968,E2 6318.968} C_VEL
LIN {X 0,Y 422.113,Z 1022.777,A -85,B 0,C 180,E1 6317.774,E2 6317.774} C_VEL
LIN {X 0,Y 431.044,Z 997.761,A -85,B 0,C 180,E1 6316.804,E2 6316.804} C_VEL
LIN {X 0,Y 437.684,Z 976.357,A -85,B 0,C 180,E1 6316.126,E2 6316.126} C_VEL
LIN {X 0,Y 443.33,Z 955.043,A -85,B 0,C 180,E1 6315.569,E2 6315.569} C_VEL
LIN {X 0,Y 448.984,Z 929.192,A -85,B 0,C 180,E1 6315.034,E2 6315.034} C_VEL
LIN {X 0,Y 453.272,Z 901.327,A -85,B 0,C 180,E1 6314.565,E2 6314.565} C_VEL
LIN {X 0,Y 462.489,Z 809.542,A -85,B 0,C 180,E1 6313.209,E2 6313.209} C_VEL
LIN {X 0,Y 475.096,Z 682.702,A -85,B 0,C 180,E1 6311.349,E2 6311.349} C_VEL
LIN {X 0,Y 472.529,Z 677.804,A -85,B 0,C 180,E1 6309.254,E2 6309.254} C_VEL
LIN {X 0,Y 471.172,Z 675.291,A -85,B 0,C 180,E1 6307.929,E2 6307.929} C_VEL
LIN {X 0,Y 469.343,Z 671.636,A -85,B 0,C 180,E1 6305.624,E2 6305.624} C_VEL
LIN {X 0,Y 467.707,Z 667.809,A -85,B 0,C 180,E1 6301.715,E2 6301.715} C_VEL
LIN {X 0,Y 467.632,Z 667.187,A -85,B 0,C 180,E1 6300.98,E2 6300.98} C_VEL
LIN {X 0,Y 467.676,Z 667.447,A -85,B 0,C 180,E1 6298.407,E2 6298.407} C_VEL
LIN {X 0,Y 469.755,Z 672.447,A -85,B 0,C 180,E1 6293.584,E2 6293.584} C_VEL
LIN {X 0,Y 472.128,Z 677.009,A -85,B 0,C 180,E1 6290.922,E2 6290.922} C_VEL
LIN {X 0,Y 474.681,Z 681.894,A -85,B 0,C 180,E1 6288.764,E2 6288.764} C_VEL
LIN {X 0,Y 475.062,Z 682.793,A -85,B 0,C 180,E1 6288.466,E2 6288.466} C_VEL
LIN {X 0,Y 453.87,Z 895.189,A -85,B 0,C 180,E1 6285.366,E2 6285.366} C_VEL
LIN {X 0,Y 450.689,Z 917.527,A -85,B 0,C 180,E1 6285.001,E2 6285.001} C_VEL
LIN {X 0,Y 445.863,Z 942.632,A -85,B 0,C 180,E1 6284.518,E2 6284.518} C_VEL
LIN {X 0,Y 439.075,Z 969.708,A -85,B 0,C 180,E1 6283.833,E2 6283.833} C_VEL
LIN {X 0,Y 432.53,Z 991.369,A -85,B 0,C 180,E1 6283.151,E2 6283.151} C_VEL
LIN {X 0,Y 425.431,Z 1011.82,A -85,B 0,C 180,E1 6282.376,E2 6282.376} C_VEL
LIN {X 0,Y 417.332,Z 1032.445,A -85,B 0,C 180,E1 6281.45,E2 6281.45} C_VEL
LIN {X 0,Y 406.679,Z 1056.548,A -85,B 0,C 180,E1 6280.151,E2 6280.151} C_VEL
LIN {X 0,Y 395.528,Z 1078.602,A -85,B 0,C 180,E1 6278.702,E2 6278.702} C_VEL
LIN {X 0,Y 385.25,Z 1097.211,A -85,B 0,C 180,E1 6277.249,E2 6277.249} C_VEL
LIN {X 0,Y 375.171,Z 1114.072,A -85,B 0,C 180,E1 6275.716,E2 6275.716} C_VEL
LIN {X 0,Y 363.764,Z 1131.812,A -85,B 0,C 180,E1 6273.831,E2 6273.831} C_VEL
LIN {X 0,Y 348.975,Z 1153.063,A -85,B 0,C 180,E1 6271.088,E2 6271.088} C_VEL
LIN {X 0,Y 337.264,Z 1168.7,A -85,B 0,C 180,E1 6268.636,E2 6268.636} C_VEL
LIN {X 0,Y 326.493,Z 1182.42,A -85,B 0,C 180,E1 6266.098,E2 6266.098} C_VEL
LIN {X 0,Y 315.791,Z 1195.53,A -85,B 0,C 180,E1 6263.238,E2 6263.238} C_VEL
LIN {X 0,Y 304.223,Z 1209.312,A -85,B 0,C 180,E1 6259.648,E2 6259.648} C_VEL
LIN {X 0,Y 292.101,Z 1223.329,A -85,B 0,C 180,E1 6255.125,E2 6255.125} C_VEL
LIN {X 0,Y 283.171,Z 1233.606,A -85,B 0,C 180,E1 6251.06,E2 6251.06} C_VEL
LIN {X 0,Y 275.919,Z 1242.179,A -85,B 0,C 180,E1 6246.987,E2 6246.987} C_VEL
LIN {X 0,Y 269.584,Z 1249.98,A -85,B 0,C 180,E1 6242.54,E2 6242.54} C_VEL
LIN {X 0,Y 263.587,Z 1258.114,A -85,B 0,C 180,E1 6236.84,E2 6236.84} C_VEL
LIN {X 0,Y 259.492,Z 1264.352,A -85,B 0,C 180,E1 6231.005,E2 6231.005} C_VEL
LIN {X 0,Y 257.469,Z 1268.273,A -85,B 0,C 180,E1 6226.243,E2 6226.243} C_VEL
LIN {X 0,Y 256.45,Z 1271.062,A -85,B 0,C 180,E1 6221.704,E2 6221.704} C_VEL
LIN {X 0,Y 256.03,Z 1272.944,A -85,B 0,C 180,E1 6217.185,E2 6217.185} C_VEL
LIN {X 0,Y 255.921,Z 1273.91,A -85,B 0,C 180,E1 6212.918,E2 6212.918} C_VEL
LIN {X 0,Y 255.899,Z 1274.079,A -85,B 0,C 180,E1 6208.663,E2 6208.663} C_VEL
LIN {X 0,Y 255.97,Z 1273.383,A -85,B 0,C 180,E1 6204.178,E2 6204.178} C_VEL
LIN {X 0,Y 256.242,Z 1271.728,A -85,B 0,C 180,E1 6199.527,E2 6199.527} C_VEL
LIN {X 0,Y 257.134,Z 1269.148,A -85,B 0,C 180,E1 6194.906,E2 6194.906} C_VEL
LIN {X 0,Y 258.878,Z 1265.482,A -85,B 0,C 180,E1 6190.138,E2 6190.138} C_VEL
LIN {X 0,Y 261.694,Z 1260.772,A -85,B 0,C 180,E1 6185.396,E2 6185.396} C_VEL
LIN {X 0,Y 265.649,Z 1255.134,A -85,B 0,C 180,E1 6180.838,E2 6180.838} C_VEL
LIN {X 0,Y 271.135,Z 1248.072,A -85,B 0,C 180,E1 6176.17,E2 6176.17} C_VEL
LIN {X 0,Y 279.644,Z 1237.934,A -85,B 0,C 180,E1 6170.747,E2 6170.747} C_VEL
LIN {X 0,Y 289.347,Z 1226.535,A -85,B 0,C 180,E1 6165.954,E2 6165.954} C_VEL
LIN {X 0,Y 298.533,Z 1215.929,A -85,B 0,C 180,E1 6162.262,E2 6162.262} C_VEL
LIN {X 0,Y 308.36,Z 1204.486,A -85,B 0,C 180,E1 6158.914,E2 6158.914} C_VEL
LIN {X 0,Y 320.877,Z 1189.61,A -85,B 0,C 180,E1 6155.285,E2 6155.285} C_VEL
LIN {X 0,Y 334.488,Z 1172.476,A -85,B 0,C 180,E1 6151.914,E2 6151.914} C_VEL
LIN {X 0,Y 345.705,Z 1157.655,A -85,B 0,C 180,E1 6149.488,E2 6149.488} C_VEL
LIN {X 0,Y 356.766,Z 1142.229,A -85,B 0,C 180,E1 6147.338,E2 6147.338} C_VEL
LIN {X 0,Y 368.286,Z 1125.152,A -85,B 0,C 180,E1 6145.316,E2 6145.316} C_VEL
LIN {X 0,Y 382.512,Z 1102.238,A -85,B 0,C 180,E1 6143.072,E2 6143.072} C_VEL
LIN {X 0,Y 393.329,Z 1083.017,A -85,B 0,C 180,E1 6141.519,E2 6141.519} C_VEL
LIN {X 0,Y 402.831,Z 1064.656,A -85,B 0,C 180,E1 6140.259,E2 6140.259} C_VEL
LIN {X 0,Y 411.72,Z 1045.772,A -85,B 0,C 180,E1 6139.139,E2 6139.139} C_VEL
LIN {X 0,Y 420.684,Z 1024.691,A -85,B 0,C 180,E1 6138.082,E2 6138.082} C_VEL
LIN {X 0,Y 430.664,Z 997.642,A -85,B 0,C 180,E1 6136.973,E2 6136.973} C_VEL
LIN {X 0,Y 437.508,Z 975.802,A -85,B 0,C 180,E1 6136.247,E2 6136.247} C_VEL
LIN {X 0,Y 439.289,Z 968.677,A -85,B 0,C 180,E1 6135.914,E2 6135.914} C_VEL
LIN {X 0,Y 442.377,Z 951.138,A -85,B 0,C 180,E1 6134.696,E2 6134.696} C_VEL
LIN {X 0,Y 443.749,Z 943.845,A -85,B 0,C 180,E1 6134.409,E2 6134.409} C_VEL
LIN {X 0,Y 448.828,Z 917.927,A -85,B 0,C 180,E1 6133.918,E2 6133.918} C_VEL
LIN {X 0,Y 452.08,Z 895.539,A -85,B 0,C 180,E1 6133.557,E2 6133.557} C_VEL
LIN {X 0,Y 473.108,Z 689.028,A -85,B 0,C 180,E1 6130.575,E2 6130.575} C_VEL
LIN {X 0,Y 471.495,Z 685.7,A -85,B 0,C 180,E1 6129.152,E2 6129.152} C_VEL
LIN {X 0,Y 470.185,Z 683.206,A -85,B 0,C 180,E1 6127.822,E2 6127.822} C_VEL
LIN {X 0,Y 468.435,Z 679.616,A -85,B 0,C 180,E1 6125.512,E2 6125.512} C_VEL
LIN {X 0,Y 466.92,Z 675.821,A -85,B 0,C 180,E1 6121.473,E2 6121.473} C_VEL
LIN {X 0,Y 466.875,Z 675.204,A -85,B 0,C 180,E1 6120.614,E2 6120.614} C_VEL
LIN {X 0,Y 466.91,Z 675.516,A -85,B 0,C 180,E1 6118.896,E2 6118.896} C_VEL
LIN {X 0,Y 468.108,Z 679.238,A -85,B 0,C 180,E1 6115.099,E2 6115.099} C_VEL
LIN {X 0,Y 468.825,Z 680.433,A -85,B 0,C 180,E1 6114.001,E2 6114.001} C_VEL
LIN {X 0,Y 471.229,Z 685.177,A -85,B 0,C 180,E1 6111.212,E2 6111.212} C_VEL
LIN {X 0,Y 473.158,Z 689.035,A -85,B 0,C 180,E1 6109.501,E2 6109.501} C_VEL
LIN {X 0,Y 452.091,Z 896.459,A -85,B 0,C 180,E1 6106.503,E2 6106.503} C_VEL
LIN {X 0,Y 448.933,Z 918.706,A -85,B 0,C 180,E1 6106.145,E2 6106.145} C_VEL
LIN {X 0,Y 444.501,Z 941.774,A -85,B 0,C 180,E1 6105.727,E2 6105.727} C_VEL
LIN {X 0,Y 437.644,Z 969.611,A -85,B 0,C 180,E1 6105.087,E2 6105.087} C_VEL
LIN {X 0,Y 430.739,Z 992.335,A -85,B 0,C 180,E1 6104.416,E2 6104.416} C_VEL
LIN {X 0,Y 423.299,Z 1013.526,A -85,B 0,C 180,E1 6103.659,E2 6103.659} C_VEL
LIN {X 0,Y 415.452,Z 1033.291,A -85,B 0,C 180,E1 6102.817,E2 6102.817} C_VEL
LIN {X 0,Y 406.291,Z 1053.952,A -85,B 0,C 180,E1 6101.775,E2 6101.775} C_VEL
LIN {X 0,Y 393.643,Z 1079.282,A -85,B 0,C 180,E1 6100.218,E2 6100.218} C_VEL
LIN {X 0,Y 382.862,Z 1098.567,A -85,B 0,C 180,E1 6098.784,E2 6098.784} C_VEL
LIN {X 0,Y 371.947,Z 1116.55,A -85,B 0,C 180,E1 6097.213,E2 6097.213} C_VEL
LIN {X 0,Y 360.593,Z 1133.931,A -85,B 0,C 180,E1 6095.421,E2 6095.421} C_VEL
LIN {X 0,Y 346.401,Z 1154.18,A -85,B 0,C 180,E1 6092.919,E2 6092.919} C_VEL
LIN {X 0,Y 332.884,Z 1171.88,A -85,B 0,C 180,E1 6090.221,E2 6090.221} C_VEL
LIN {X 0,Y 321.716,Z 1185.824,A -85,B 0,C 180,E1 6087.685,E2 6087.685} C_VEL
LIN {X 0,Y 310.558,Z 1199.194,A -85,B 0,C 180,E1 6084.808,E2 6084.808} C_VEL
LIN {X 0,Y 298.67,Z 1213,A -85,B 0,C 180,E1 6081.252,E2 6081.252} C_VEL
LIN {X 0,Y 285.453,Z 1227.908,A -85,B 0,C 180,E1 6076.464,E2 6076.464} C_VEL
LIN {X 0,Y 276.187,Z 1238.333,A -85,B 0,C 180,E1 6072.318,E2 6072.318} C_VEL
LIN {X 0,Y 268.597,Z 1247.044,A -85,B 0,C 180,E1 6068.157,E2 6068.157} C_VEL
LIN {X 0,Y 261.71,Z 1255.338,A -85,B 0,C 180,E1 6063.369,E2 6063.369} C_VEL
LIN {X 0,Y 255.139,Z 1264.036,A -85,B 0,C 180,E1 6057.031,E2 6057.031} C_VEL
LIN {X 0,Y 251.347,Z 1269.841,A -85,B 0,C 180,E1 6051.46,E2 6051.46} C_VEL
LIN {X 0,Y 249.39,Z 1273.647,A -85,B 0,C 180,E1 6046.771,E2 6046.771} C_VEL
LIN {X 0,Y 248.369,Z 1276.508,A -85,B 0,C 180,E1 6042.076,E2 6042.076} C_VEL
LIN {X 0,Y 247.982,Z 1278.438,A -85,B 0,C 180,E1 6037.406,E2 6037.406} C_VEL
LIN {X 0,Y 247.913,Z 1279.424,A -85,B 0,C 180,E1 6032.999,E2 6032.999} C_VEL
LIN {X 0,Y 247.902,Z 1279.581,A -85,B 0,C 180,E1 6028.607,E2 6028.607} C_VEL
LIN {X 0,Y 247.943,Z 1278.843,A -85,B 0,C 180,E1 6023.975,E2 6023.975} C_VEL
LIN {X 0,Y 248.174,Z 1277.181,A -85,B 0,C 180,E1 6019.313,E2 6019.313} C_VEL
LIN {X 0,Y 249.07,Z 1274.431,A -85,B 0,C 180,E1 6014.391,E2 6014.391} C_VEL
LIN {X 0,Y 250.893,Z 1270.644,A -85,B 0,C 180,E1 6009.463,E2 6009.463} C_VEL
LIN {X 0,Y 253.857,Z 1265.794,A -85,B 0,C 180,E1 6004.569,E2 6004.569} C_VEL
LIN {X 0,Y 258.109,Z 1259.851,A -85,B 0,C 180,E1 5999.755,E2 5999.755} C_VEL
LIN {X 0,Y 264.346,Z 1252.062,A -85,B 0,C 180,E1 5994.634,E2 5994.634} C_VEL
LIN {X 0,Y 274.177,Z 1240.563,A -85,B 0,C 180,E1 5988.688,E2 5988.688} C_VEL
LIN {X 0,Y 283.155,Z 1230.409,A -85,B 0,C 180,E1 5984.49,E2 5984.49} C_VEL
LIN {X 0,Y 292.372,Z 1220.026,A -85,B 0,C 180,E1 5980.899,E2 5980.899} C_VEL
LIN {X 0,Y 303.123,Z 1207.763,A -85,B 0,C 180,E1 5977.342,E2 5977.342} C_VEL
LIN {X 0,Y 316.84,Z 1191.711,A -85,B 0,C 180,E1 5973.523,E2 5973.523} C_VEL
LIN {X 0,Y 330.231,Z 1175.095,A -85,B 0,C 180,E1 5970.347,E2 5970.347} C_VEL
LIN {X 0,Y 341.839,Z 1160.021,A -85,B 0,C 180,E1 5967.945,E2 5967.945} C_VEL
LIN {X 0,Y 353.268,Z 1144.339,A -85,B 0,C 180,E1 5965.828,E2 5965.828} C_VEL
LIN {X 0,Y 367.071,Z 1124.141,A -85,B 0,C 180,E1 5963.542,E2 5963.542} C_VEL
LIN {X 0,Y 379.932,Z 1103.292,A -85,B 0,C 180,E1 5961.62,E2 5961.62} C_VEL
LIN {X 0,Y 390.038,Z 1085.548,A -85,B 0,C 180,E1 5960.233,E2 5960.233} C_VEL
LIN {X 0,Y 399.749,Z 1067.033,A -85,B 0,C 180,E1 5959.001,E2 5959.001} C_VEL
LIN {X 0,Y 409.08,Z 1047.495,A -85,B 0,C 180,E1 5957.891,E2 5957.891} C_VEL
LIN {X 0,Y 419.424,Z 1023.391,A -85,B 0,C 180,E1 5956.748,E2 5956.748} C_VEL
LIN {X 0,Y 428.626,Z 998.113,A -85,B 0,C 180,E1 5955.784,E2 5955.784} C_VEL
LIN {X 0,Y 435.295,Z 977,A -85,B 0,C 180,E1 5955.127,E2 5955.127} C_VEL
LIN {X 0,Y 441,Z 955.89,A -85,B 0,C 180,E1 5954.583,E2 5954.583} C_VEL
LIN {X 0,Y 446.225,Z 932.615,A -85,B 0,C 180,E1 5954.105,E2 5954.105} C_VEL
LIN {X 0,Y 451.16,Z 902.524,A -85,B 0,C 180,E1 5953.597,E2 5953.597} C_VEL
LIN {X 0,Y 457.903,Z 837.584,A -85,B 0,C 180,E1 5952.642,E2 5952.642} C_VEL
LIN {X 0,Y 472.954,Z 688.818,A -85,B 0,C 180,E1 5950.494,E2 5950.494} C_VEL
LIN {X 0,Y 470.433,Z 683.704,A -85,B 0,C 180,E1 5948.187,E2 5948.187} C_VEL
LIN {X 0,Y 468.281,Z 679.516,A -85,B 0,C 180,E1 5945.514,E2 5945.514} C_VEL
LIN {X 0,Y 466.71,Z 675.69,A -85,B 0,C 180,E1 5941.596,E2 5941.596} C_VEL
LIN {X 0,Y 466.639,Z 675.13,A -85,B 0,C 180,E1 5940.859,E2 5940.859} C_VEL
LIN {X 0,Y 466.684,Z 675.329,A -85,B 0,C 180,E1 5938.527,E2 5938.527} C_VEL
LIN {X 0,Y 468.64,Z 680.251,A -85,B 0,C 180,E1 5933.753,E2 5933.753} C_VEL
LIN {X 0,Y 470.887,Z 684.698,A -85,B 0,C 180,E1 5931.144,E2 5931.144} C_VEL
LIN {X 0,Y 472.923,Z 688.729,A -85,B 0,C 180,E1 5929.334,E2 5929.334} C_VEL
LIN {X 0,Y 451.708,Z 896.969,A -85,B 0,C 180,E1 5926.325,E2 5926.325} C_VEL
LIN {X 0,Y 448.152,Z 920.826,A -85,B 0,C 180,E1 5925.936,E2 5925.936} C_VEL
LIN {X 0,Y 442.035,Z 950.129,A -85,B 0,C 180,E1 5925.349,E2 5925.349} C_VEL
LIN {X 0,Y 436.255,Z 972.021,A -85,B 0,C 180,E1 5924.784,E2 5924.784} C_VEL
LIN {X 0,Y 429.834,Z 992.748,A -85,B 0,C 180,E1 5924.136,E2 5924.136} C_VEL
LIN {X 0,Y 422.484,Z 1013.436,A -85,B 0,C 180,E1 5923.359,E2 5923.359} C_VEL
LIN {X 0,Y 412.596,Z 1037.92,A -85,B 0,C 180,E1 5922.255,E2 5922.255} C_VEL
LIN {X 0,Y 401.532,Z 1061.495,A -85,B 0,C 180,E1 5920.94,E2 5920.94} C_VEL
LIN {X 0,Y 391.62,Z 1080.545,A -85,B 0,C 180,E1 5919.681,E2 5919.681} C_VEL
LIN {X 0,Y 381.752,Z 1097.986,A -85,B 0,C 180,E1 5918.327,E2 5918.327} C_VEL
LIN {X 0,Y 371.477,Z 1114.773,A -85,B 0,C 180,E1 5916.814,E2 5916.814} C_VEL
LIN {X 0,Y 358.702,Z 1134.155,A -85,B 0,C 180,E1 5914.755,E2 5914.755} C_VEL
LIN {X 0,Y 344.684,Z 1153.618,A -85,B 0,C 180,E1 5912.228,E2 5912.228} C_VEL
LIN {X 0,Y 333.003,Z 1168.795,A -85,B 0,C 180,E1 5909.861,E2 5909.861} C_VEL
LIN {X 0,Y 321.546,Z 1182.954,A -85,B 0,C 180,E1 5907.243,E2 5907.243} C_VEL
LIN {X 0,Y 310.264,Z 1196.32,A -85,B 0,C 180,E1 5904.309,E2 5904.309} C_VEL
LIN {X 0,Y 296.907,Z 1211.654,A -85,B 0,C 180,E1 5900.218,E2 5900.218} C_VEL
LIN {X 0,Y 285.303,Z 1224.444,A -85,B 0,C 180,E1 5895.933,E2 5895.933} C_VEL
LIN {X 0,Y 276.499,Z 1234.154,A -85,B 0,C 180,E1 5891.996,E2 5891.996} C_VEL
LIN {X 0,Y 268.584,Z 1243.074,A -85,B 0,C 180,E1 5887.634,E2 5887.634} C_VEL
LIN {X 0,Y 260.664,Z 1252.51,A -85,B 0,C 180,E1 5881.968,E2 5881.968} C_VEL
LIN {X 0,Y 254.822,Z 1259.973,A -85,B 0,C 180,E1 5876.076,E2 5876.076} C_VEL
LIN {X 0,Y 251.56,Z 1264.85,A -85,B 0,C 180,E1 5871.211,E2 5871.211} C_VEL
LIN {X 0,Y 249.548,Z 1268.52,A -85,B 0,C 180,E1 5866.534,E2 5866.534} C_VEL
LIN {X 0,Y 248.471,Z 1271.263,A -85,B 0,C 180,E1 5861.849,E2 5861.849} C_VEL
LIN {X 0,Y 248.04,Z 1273.037,A -85,B 0,C 180,E1 5857.4,E2 5857.4} C_VEL
LIN {X 0,Y 247.922,Z 1273.998,A -85,B 0,C 180,E1 5853.012,E2 5853.012} C_VEL
LIN {X 0,Y 247.901,Z 1274.167,A -85,B 0,C 180,E1 5848.62,E2 5848.62} C_VEL
LIN {X 0,Y 247.978,Z 1273.471,A -85,B 0,C 180,E1 5843.989,E2 5843.989} C_VEL
LIN {X 0,Y 248.268,Z 1271.884,A -85,B 0,C 180,E1 5839.329,E2 5839.329} C_VEL
LIN {X 0,Y 249.289,Z 1269.151,A -85,B 0,C 180,E1 5834.289,E2 5834.289} C_VEL
LIN {X 0,Y 251.156,Z 1265.572,A -85,B 0,C 180,E1 5829.5,E2 5829.5} C_VEL
LIN {X 0,Y 254.191,Z 1260.862,A -85,B 0,C 180,E1 5824.619,E2 5824.619} C_VEL
LIN {X 0,Y 258.528,Z 1255.073,A -85,B 0,C 180,E1 5819.824,E2 5819.824} C_VEL
LIN {X 0,Y 264.531,Z 1247.812,A -85,B 0,C 180,E1 5814.942,E2 5814.942} C_VEL
LIN {X 0,Y 273.963,Z 1237.114,A -85,B 0,C 180,E1 5809.219,E2 5809.219} C_VEL
LIN {X 0,Y 283.737,Z 1226.229,A -85,B 0,C 180,E1 5804.626,E2 5804.626} C_VEL
LIN {X 0,Y 293.567,Z 1215.36,A -85,B 0,C 180,E1 5800.841,E2 5800.841} C_VEL
LIN {X 0,Y 304.872,Z 1202.683,A -85,B 0,C 180,E1 5797.171,E2 5797.171} C_VEL
LIN {X 0,Y 319.325,Z 1185.811,A -85,B 0,C 180,E1 5793.228,E2 5793.228} C_VEL
LIN {X 0,Y 331.475,Z 1170.882,A -85,B 0,C 180,E1 5790.392,E2 5790.392} C_VEL
LIN {X 0,Y 343.084,Z 1155.899,A -85,B 0,C 180,E1 5788.001,E2 5788.001} C_VEL
LIN {X 0,Y 355.23,Z 1139.288,A -85,B 0,C 180,E1 5785.763,E2 5785.763} C_VEL
LIN {X 0,Y 370.138,Z 1117.158,A -85,B 0,C 180,E1 5783.314,E2 5783.314} C_VEL
LIN {X 0,Y 381.432,Z 1098.809,A -85,B 0,C 180,E1 5781.637,E2 5781.637} C_VEL
LIN {X 0,Y 391.596,Z 1080.904,A -85,B 0,C 180,E1 5780.241,E2 5780.241} C_VEL
LIN {X 0,Y 401.288,Z 1062.328,A -85,B 0,C 180,E1 5779.011,E2 5779.011} C_VEL
LIN {X 0,Y 411.986,Z 1039.662,A -85,B 0,C 180,E1 5777.734,E2 5777.734} C_VEL
LIN {X 0,Y 422.023,Z 1015.166,A -85,B 0,C 180,E1 5776.613,E2 5776.613} C_VEL
LIN {X 0,Y 429.704,Z 993.703,A -85,B 0,C 180,E1 5775.798,E2 5775.798} C_VEL
LIN {X 0,Y 436.101,Z 973.204,A -85,B 0,C 180,E1 5775.152,E2 5775.152} C_VEL
LIN {X 0,Y 441.893,Z 951.465,A -85,B 0,C 180,E1 5774.585,E2 5774.585} C_VEL
LIN {X 0,Y 443.749,Z 943.845,A -85,B 0,C 180,E1 5774.409,E2 5774.409} C_VEL
LIN {X 0,Y 445.074,Z 936.481,A -85,B 0,C 180,E1 5774.137,E2 5774.137} C_VEL
LIN {X 0,Y 447.268,Z 917.292,A -85,B 0,C 180,E1 5773.004,E2 5773.004} C_VEL
LIN {X 0,Y 448.159,Z 910.898,A -85,B 0,C 180,E1 5772.802,E2 5772.802} C_VEL
LIN {X 0,Y 452.541,Z 875.102,A -85,B 0,C 180,E1 5772.262,E2 5772.262} C_VEL
LIN {X 0,Y 471.071,Z 694.908,A -85,B 0,C 180,E1 5769.684,E2 5769.684} C_VEL
LIN {X 0,Y 469.091,Z 691.095,A -85,B 0,C 180,E1 5767.717,E2 5767.717} C_VEL
LIN {X 0,Y 467.377,Z 687.497,A -85,B 0,C 180,E1 5765.401,E2 5765.401} C_VEL
LIN {X 0,Y 465.929,Z 683.701,A -85,B 0,C 180,E1 5761.353,E2 5761.353} C_VEL
LIN {X 0,Y 465.891,Z 683.15,A -85,B 0,C 180,E1 5760.492,E2 5760.492} C_VEL
LIN {X 0,Y 465.923,Z 683.395,A -85,B 0,C 180,E1 5759.016,E2 5759.016} C_VEL
LIN {X 0,Y 467.131,Z 687.219,A -85,B 0,C 180,E1 5755.088,E2 5755.088} C_VEL
LIN {X 0,Y 467.793,Z 688.455,A -85,B 0,C 180,E1 5754.05,E2 5754.05} C_VEL
LIN {X 0,Y 469.992,Z 692.865,A -85,B 0,C 180,E1 5751.435,E2 5751.435} C_VEL
LIN {X 0,Y 471.098,Z 695.307,A -85,B 0,C 180,E1 5750.37,E2 5750.37} C_VEL
LIN {X 0,Y 449.875,Z 899.714,A -85,B 0,C 180,E1 5747.447,E2 5747.447} C_VEL
LIN {X 0,Y 446.062,Z 924.684,A -85,B 0,C 180,E1 5747.045,E2 5747.045} C_VEL
LIN {X 0,Y 439.895,Z 953.22,A -85,B 0,C 180,E1 5746.499,E2 5746.499} C_VEL
LIN {X 0,Y 434.122,Z 974.643,A -85,B 0,C 180,E1 5745.974,E2 5745.974} C_VEL
LIN {X 0,Y 427.767,Z 994.827,A -85,B 0,C 180,E1 5745.374,E2 5745.374} C_VEL
LIN {X 0,Y 420.406,Z 1015.238,A -85,B 0,C 180,E1 5744.649,E2 5744.649} C_VEL
LIN {X 0,Y 411.423,Z 1037.235,A -85,B 0,C 180,E1 5743.711,E2 5743.711} C_VEL
LIN {X 0,Y 399.361,Z 1062.986,A -85,B 0,C 180,E1 5742.365,E2 5742.365} C_VEL
LIN {X 0,Y 388.886,Z 1082.88,A -85,B 0,C 180,E1 5741.097,E2 5741.097} C_VEL
LIN {X 0,Y 379.156,Z 1099.821,A -85,B 0,C 180,E1 5739.835,E2 5739.835} C_VEL
LIN {X 0,Y 368.442,Z 1117.059,A -85,B 0,C 180,E1 5738.341,E2 5738.341} C_VEL
LIN {X 0,Y 356.464,Z 1134.958,A -85,B 0,C 180,E1 5736.508,E2 5736.508} C_VEL
LIN {X 0,Y 340.866,Z 1156.416,A -85,B 0,C 180,E1 5733.83,E2 5733.83} C_VEL
LIN {X 0,Y 328.122,Z 1172.641,A -85,B 0,C 180,E1 5731.342,E2 5731.342} C_VEL
LIN {X 0,Y 316.675,Z 1186.492,A -85,B 0,C 180,E1 5728.813,E2 5728.813} C_VEL
LIN {X 0,Y 305.161,Z 1199.832,A -85,B 0,C 180,E1 5725.923,E2 5725.923} C_VEL
LIN {X 0,Y 291.801,Z 1214.826,A -85,B 0,C 180,E1 5721.998,E2 5721.998} C_VEL
LIN {X 0,Y 279.221,Z 1228.336,A -85,B 0,C 180,E1 5717.523,E2 5717.523} C_VEL
LIN {X 0,Y 269.823,Z 1238.463,A -85,B 0,C 180,E1 5713.421,E2 5713.421} C_VEL
LIN {X 0,Y 261.676,Z 1247.362,A -85,B 0,C 180,E1 5709.075,E2 5709.075} C_VEL
LIN {X 0,Y 253.886,Z 1256.317,A -85,B 0,C 180,E1 5703.722,E2 5703.722} C_VEL
LIN {X 0,Y 247.345,Z 1264.46,A -85,B 0,C 180,E1 5697.433,E2 5697.433} C_VEL
LIN {X 0,Y 243.679,Z 1269.751,A -85,B 0,C 180,E1 5692.171,E2 5692.171} C_VEL
LIN {X 0,Y 241.555,Z 1273.558,A -85,B 0,C 180,E1 5687.332,E2 5687.332} C_VEL
LIN {X 0,Y 240.423,Z 1276.419,A -85,B 0,C 180,E1 5682.482,E2 5682.482} C_VEL
LIN {X 0,Y 239.982,Z 1278.35,A -85,B 0,C 180,E1 5677.655,E2 5677.655} C_VEL
LIN {X 0,Y 239.914,Z 1279.313,A -85,B 0,C 180,E1 5673.338,E2 5673.338} C_VEL
LIN {X 0,Y 239.893,Z 1279.517,A -85,B 0,C 180,E1 5668.799,E2 5668.799} C_VEL
LIN {X 0,Y 239.942,Z 1278.823,A -85,B 0,C 180,E1 5664.013,E2 5664.013} C_VEL
LIN {X 0,Y 240.219,Z 1277.092,A -85,B 0,C 180,E1 5658.955,E2 5658.955} C_VEL
LIN {X 0,Y 241.19,Z 1274.341,A -85,B 0,C 180,E1 5653.867,E2 5653.867} C_VEL
LIN {X 0,Y 243.177,Z 1270.553,A -85,B 0,C 180,E1 5648.781,E2 5648.781} C_VEL
LIN {X 0,Y 246.39,Z 1265.703,A -85,B 0,C 180,E1 5643.741,E2 5643.741} C_VEL
LIN {X 0,Y 250.932,Z 1259.758,A -85,B 0,C 180,E1 5638.795,E2 5638.795} C_VEL
LIN {X 0,Y 257.226,Z 1252.325,A -85,B 0,C 180,E1 5633.776,E2 5633.776} C_VEL
LIN {X 0,Y 267.502,Z 1240.932,A -85,B 0,C 180,E1 5627.709,E2 5627.709} C_VEL
LIN {X 0,Y 277.317,Z 1230.316,A -85,B 0,C 180,E1 5623.248,E2 5623.248} C_VEL
LIN {X 0,Y 286.954,Z 1219.903,A -85,B 0,C 180,E1 5619.618,E2 5619.618} C_VEL
LIN {X 0,Y 298.095,Z 1207.669,A -85,B 0,C 180,E1 5616.057,E2 5616.057} C_VEL
LIN {X 0,Y 312.182,Z 1191.733,A -85,B 0,C 180,E1 5612.262,E2 5612.262} C_VEL
LIN {X 0,Y 325.401,Z 1175.85,A -85,B 0,C 180,E1 5609.224,E2 5609.224} C_VEL
LIN {X 0,Y 337.292,Z 1160.856,A -85,B 0,C 180,E1 5606.831,E2 5606.831} C_VEL
LIN {X 0,Y 348.982,Z 1145.26,A -85,B 0,C 180,E1 5604.728,E2 5604.728} C_VEL
LIN {X 0,Y 360.544,Z 1128.81,A -85,B 0,C 180,E1 5602.846,E2 5602.846} C_VEL
LIN {X 0,Y 374.76,Z 1106.923,A -85,B 0,C 180,E1 5600.762,E2 5600.762} C_VEL
LIN {X 0,Y 386.644,Z 1086.596,A -85,B 0,C 180,E1 5599.174,E2 5599.174} C_VEL
LIN {X 0,Y 396.785,Z 1067.671,A -85,B 0,C 180,E1 5597.928,E2 5597.928} C_VEL
LIN {X 0,Y 405.903,Z 1048.992,A -85,B 0,C 180,E1 5596.879,E2 5596.879} C_VEL
LIN {X 0,Y 414.864,Z 1028.672,A -85,B 0,C 180,E1 5595.913,E2 5595.913} C_VEL
LIN {X 0,Y 424.764,Z 1003.164,A -85,B 0,C 180,E1 5594.91,E2 5594.91} C_VEL
LIN {X 0,Y 432.718,Z 978.733,A -85,B 0,C 180,E1 5594.147,E2 5594.147} C_VEL
LIN {X 0,Y 438.694,Z 957.158,A -85,B 0,C 180,E1 5593.597,E2 5593.597} C_VEL
LIN {X 0,Y 443.73,Z 935.354,A -85,B 0,C 180,E1 5593.151,E2 5593.151} C_VEL
LIN {X 0,Y 448.632,Z 908.114,A -85,B 0,C 180,E1 5592.688,E2 5592.688} C_VEL
LIN {X 0,Y 453.485,Z 864.352,A -85,B 0,C 180,E1 5592.042,E2 5592.042} C_VEL
LIN {X 0,Y 470.922,Z 694.832,A -85,B 0,C 180,E1 5589.626,E2 5589.626} C_VEL
LIN {X 0,Y 468.864,Z 690.889,A -85,B 0,C 180,E1 5587.598,E2 5587.598} C_VEL
LIN {X 0,Y 467.138,Z 687.296,A -85,B 0,C 180,E1 5585.281,E2 5585.281} C_VEL
LIN {X 0,Y 465.714,Z 683.57,A -85,B 0,C 180,E1 5581.476,E2 5581.476} C_VEL
LIN {X 0,Y 465.648,Z 683.074,A -85,B 0,C 180,E1 5580.738,E2 5580.738} C_VEL
LIN {X 0,Y 465.694,Z 683.21,A -85,B 0,C 180,E1 5578.647,E2 5578.647} C_VEL
LIN {X 0,Y 467.529,Z 688.055,A -85,B 0,C 180,E1 5573.923,E2 5573.923} C_VEL
LIN {X 0,Y 469.712,Z 692.52,A -85,B 0,C 180,E1 5571.307,E2 5571.307} C_VEL
LIN {X 0,Y 470.864,Z 694.944,A -85,B 0,C 180,E1 5570.207,E2 5570.207} C_VEL
LIN {X 0,Y 449.832,Z 897.464,A -85,B 0,C 180,E1 5567.311,E2 5567.311} C_VEL
LIN {X 0,Y 446.045,Z 922.278,A -85,B 0,C 180,E1 5566.913,E2 5566.913} C_VEL
LIN {X 0,Y 439.944,Z 950.729,A -85,B 0,C 180,E1 5566.35,E2 5566.35} C_VEL
LIN {X 0,Y 433.993,Z 972.857,A -85,B 0,C 180,E1 5565.789,E2 5565.789} C_VEL
LIN {X 0,Y 427.698,Z 992.845,A -85,B 0,C 180,E1 5565.176,E2 5565.176} C_VEL
LIN {X 0,Y 420.386,Z 1013.139,A -85,B 0,C 180,E1 5564.432,E2 5564.432} C_VEL
LIN {X 0,Y 411.036,Z 1036.011,A -85,B 0,C 180,E1 5563.43,E2 5563.43} C_VEL
LIN {X 0,Y 399.315,Z 1060.861,A -85,B 0,C 180,E1 5562.092,E2 5562.092} C_VEL
LIN {X 0,Y 389.167,Z 1080.082,A -85,B 0,C 180,E1 5560.85,E2 5560.85} C_VEL
LIN {X 0,Y 378.966,Z 1097.803,A -85,B 0,C 180,E1 5559.502,E2 5559.502} C_VEL
LIN {X 0,Y 368.368,Z 1114.778,A -85,B 0,C 180,E1 5558.001,E2 5558.001} C_VEL
LIN {X 0,Y 355.433,Z 1133.982,A -85,B 0,C 180,E1 5555.992,E2 5555.992} C_VEL
LIN {X 0,Y 340.46,Z 1154.266,A -85,B 0,C 180,E1 5553.383,E2 5553.383} C_VEL
LIN {X 0,Y 328.213,Z 1169.729,A -85,B 0,C 180,E1 5550.972,E2 5550.972} C_VEL
LIN {X 0,Y 316.18,Z 1184.14,A -85,B 0,C 180,E1 5548.292,E2 5548.292} C_VEL
LIN {X 0,Y 302.451,Z 1199.895,A -85,B 0,C 180,E1 5544.749,E2 5544.749} C_VEL
LIN {X 0,Y 288.789,Z 1214.694,A -85,B 0,C 180,E1 5540.549,E2 5540.549} C_VEL
LIN {X 0,Y 278.564,Z 1225.559,A -85,B 0,C 180,E1 5536.78,E2 5536.78} C_VEL
LIN {X 0,Y 269.268,Z 1235.38,A -85,B 0,C 180,E1 5532.672,E2 5532.672} C_VEL
LIN {X 0,Y 259.54,Z 1245.966,A -85,B 0,C 180,E1 5527.224,E2 5527.224} C_VEL
LIN {X 0,Y 251.694,Z 1254.738,A -85,B 0,C 180,E1 5521.337,E2 5521.337} C_VEL
LIN {X 0,Y 247.012,Z 1260.567,A -85,B 0,C 180,E1 5516.447,E2 5516.447} C_VEL
LIN {X 0,Y 243.631,Z 1265.348,A -85,B 0,C 180,E1 5511.43,E2 5511.43} C_VEL
LIN {X 0,Y 241.556,Z 1268.925,A -85,B 0,C 180,E1 5506.602,E2 5506.602} C_VEL
LIN {X 0,Y 240.454,Z 1271.575,A -85,B 0,C 180,E1 5501.763,E2 5501.763} C_VEL
LIN {X 0,Y 240.032,Z 1273.254,A -85,B 0,C 180,E1 5497.186,E2 5497.186} C_VEL
LIN {X 0,Y 239.921,Z 1274.108,A -85,B 0,C 180,E1 5492.873,E2 5492.873} C_VEL
LIN {X 0,Y 239.902,Z 1274.254,A -85,B 0,C 180,E1 5488.574,E2 5488.574} C_VEL
LIN {X 0,Y 239.988,Z 1273.559,A -85,B 0,C 180,E1 5483.788,E2 5483.788} C_VEL
LIN {X 0,Y 240.354,Z 1271.861,A -85,B 0,C 180,E1 5478.732,E2 5478.732} C_VEL
LIN {X 0,Y 241.386,Z 1269.325,A -85,B 0,C 180,E1 5473.895,E2 5473.895} C_VEL
LIN {X 0,Y 243.478,Z 1265.63,A -85,B 0,C 180,E1 5468.785,E2 5468.785} C_VEL
LIN {X 0,Y 246.741,Z 1260.951,A -85,B 0,C 180,E1 5463.796,E2 5463.796} C_VEL
LIN {X 0,Y 251.365,Z 1255.163,A -85,B 0,C 180,E1 5458.87,E2 5458.87} C_VEL
LIN {X 0,Y 257.73,Z 1247.903,A -85,B 0,C 180,E1 5453.874,E2 5453.874} C_VEL
LIN {X 0,Y 267.755,Z 1237.103,A -85,B 0,C 180,E1 5448,E2 5448} C_VEL
LIN {X 0,Y 277.915,Z 1226.319,A -85,B 0,C 180,E1 5443.396,E2 5443.396} C_VEL
LIN {X 0,Y 288.075,Z 1215.539,A -85,B 0,C 180,E1 5439.609,E2 5439.609} C_VEL
LIN {X 0,Y 299.296,Z 1203.403,A -85,B 0,C 180,E1 5436.066,E2 5436.066} C_VEL
LIN {X 0,Y 314.701,Z 1186.042,A -85,B 0,C 180,E1 5431.984,E2 5431.984} C_VEL
LIN {X 0,Y 326.654,Z 1171.811,A -85,B 0,C 180,E1 5429.278,E2 5429.278} C_VEL
LIN {X 0,Y 338.546,Z 1156.909,A -85,B 0,C 180,E1 5426.897,E2 5426.897} C_VEL
LIN {X 0,Y 350.218,Z 1141.394,A -85,B 0,C 180,E1 5424.8,E2 5424.8} C_VEL
LIN {X 0,Y 363.863,Z 1122.007,A -85,B 0,C 180,E1 5422.602,E2 5422.602} C_VEL
LIN {X 0,Y 377.381,Z 1100.734,A -85,B 0,C 180,E1 5420.634,E2 5420.634} C_VEL
LIN {X 0,Y 388.077,Z 1082.364,A -85,B 0,C 180,E1 5419.207,E2 5419.207} C_VEL
LIN {X 0,Y 397.816,Z 1064.15,A -85,B 0,C 180,E1 5418.008,E2 5418.008} C_VEL
LIN {X 0,Y 407.051,Z 1045.135,A -85,B 0,C 180,E1 5416.93,E2 5416.93} C_VEL
LIN {X 0,Y 417.185,Z 1021.932,A -85,B 0,C 180,E1 5415.83,E2 5415.83} C_VEL
LIN {X 0,Y 426.656,Z 996.52,A -85,B 0,C 180,E1 5414.85,E2 5414.85} C_VEL
LIN {X 0,Y 433.401,Z 975.534,A -85,B 0,C 180,E1 5414.189,E2 5414.189} C_VEL
LIN {X 0,Y 439.199,Z 954.456,A -85,B 0,C 180,E1 5413.64,E2 5413.64} C_VEL
LIN {X 0,Y 444.138,Z 932.912,A -85,B 0,C 180,E1 5413.183,E2 5413.183} C_VEL
LIN {X 0,Y 448.159,Z 910.898,A -85,B 0,C 180,E1 5412.802,E2 5412.802} C_VEL
LIN {X 0,Y 449.025,Z 904.477,A -85,B 0,C 180,E1 5412.606,E2 5412.606} C_VEL
LIN {X 0,Y 450.157,Z 883.946,A -85,B 0,C 180,E1 5411.486,E2 5411.486} C_VEL
LIN {X 0,Y 450.668,Z 877.469,A -85,B 0,C 180,E1 5411.298,E2 5411.298} C_VEL
LIN {X 0,Y 469.119,Z 701.297,A -85,B 0,C 180,E1 5408.812,E2 5408.812} C_VEL
LIN {X 0,Y 467.783,Z 698.627,A -85,B 0,C 180,E1 5407.369,E2 5407.369} C_VEL
LIN {X 0,Y 466.243,Z 695.28,A -85,B 0,C 180,E1 5405.168,E2 5405.168} C_VEL
LIN {X 0,Y 464.938,Z 691.441,A -85,B 0,C 180,E1 5401.109,E2 5401.109} C_VEL
LIN {X 0,Y 464.901,Z 691.105,A -85,B 0,C 180,E1 5400.123,E2 5400.123} C_VEL
LIN {X 0,Y 464.938,Z 691.422,A -85,B 0,C 180,E1 5399.014,E2 5399.014} C_VEL
LIN {X 0,Y 466.231,Z 695.298,A -85,B 0,C 180,E1 5394.955,E2 5394.955} C_VEL
LIN {X 0,Y 467.092,Z 697.299,A -85,B 0,C 180,E1 5393.609,E2 5393.609} C_VEL
LIN {X 0,Y 468.82,Z 700.683,A -85,B 0,C 180,E1 5391.599,E2 5391.599} C_VEL
LIN {X 0,Y 469.148,Z 701.533,A -85,B 0,C 180,E1 5391.25,E2 5391.25} C_VEL
LIN {X 0,Y 448.183,Z 899.755,A -85,B 0,C 180,E1 5388.448,E2 5388.448} C_VEL
LIN {X 0,Y 444.235,Z 925.164,A -85,B 0,C 180,E1 5388.046,E2 5388.046} C_VEL
LIN {X 0,Y 438.037,Z 953.328,A -85,B 0,C 180,E1 5387.518,E2 5387.518} C_VEL
LIN {X 0,Y 431.993,Z 975.378,A -85,B 0,C 180,E1 5386.99,E2 5386.99} C_VEL
LIN {X 0,Y 425.356,Z 996.031,A -85,B 0,C 180,E1 5386.386,E2 5386.386} C_VEL
LIN {X 0,Y 417.46,Z 1017.42,A -85,B 0,C 180,E1 5385.634,E2 5385.634} C_VEL
LIN {X 0,Y 406.336,Z 1043.58,A -85,B 0,C 180,E1 5384.503,E2 5384.503} C_VEL
LIN {X 0,Y 395.957,Z 1064.826,A -85,B 0,C 180,E1 5383.378,E2 5383.378} C_VEL
LIN {X 0,Y 385.879,Z 1083.552,A -85,B 0,C 180,E1 5382.196,E2 5382.196} C_VEL
LIN {X 0,Y 375.58,Z 1101.074,A -85,B 0,C 180,E1 5380.905,E2 5380.905} C_VEL
LIN {X 0,Y 363.472,Z 1120.038,A -85,B 0,C 180,E1 5379.259,E2 5379.259} C_VEL
LIN {X 0,Y 347.458,Z 1142.865,A -85,B 0,C 180,E1 5376.825,E2 5376.825} C_VEL
LIN {X 0,Y 334.681,Z 1159.583,A -85,B 0,C 180,E1 5374.637,E2 5374.637} C_VEL
LIN {X 0,Y 322.402,Z 1174.704,A -85,B 0,C 180,E1 5372.276,E2 5372.276} C_VEL
LIN {X 0,Y 309.079,Z 1190.262,A -85,B 0,C 180,E1 5369.36,E2 5369.36} C_VEL
LIN {X 0,Y 293.803,Z 1207.069,A -85,B 0,C 180,E1 5365.432,E2 5365.432} C_VEL
LIN {X 0,Y 282.155,Z 1219.375,A -85,B 0,C 180,E1 5361.867,E2 5361.867} C_VEL
LIN {X 0,Y 271.588,Z 1230.32,A -85,B 0,C 180,E1 5358.035,E2 5358.035} C_VEL
LIN {X 0,Y 261.329,Z 1240.927,A -85,B 0,C 180,E1 5353.517,E2 5353.517} C_VEL
LIN {X 0,Y 250.497,Z 1252.303,A -85,B 0,C 180,E1 5347.343,E2 5347.343} C_VEL
LIN {X 0,Y 243.813,Z 1259.724,A -85,B 0,C 180,E1 5342.208,E2 5342.208} C_VEL
LIN {X 0,Y 238.958,Z 1265.657,A -85,B 0,C 180,E1 5337.126,E2 5337.126} C_VEL
LIN {X 0,Y 235.357,Z 1270.708,A -85,B 0,C 180,E1 5331.683,E2 5331.683} C_VEL
LIN {X 0,Y 233.064,Z 1274.928,A -85,B 0,C 180,E1 5325.673,E2 5325.673} C_VEL
LIN {X 0,Y 232.069,Z 1277.859,A -85,B 0,C 180,E1 5319.365,E2 5319.365} C_VEL
LIN {X 0,Y 231.917,Z 1279.178,A -85,B 0,C 180,E1 5313.948,E2 5313.948} C_VEL
LIN {X 0,Y 231.887,Z 1279.452,A -85,B 0,C 180,E1 5309.005,E2 5309.005} C_VEL
LIN {X 0,Y 231.94,Z 1278.804,A -85,B 0,C 180,E1 5304.054,E2 5304.054} C_VEL
LIN {X 0,Y 232.27,Z 1277.003,A -85,B 0,C 180,E1 5298.572,E2 5298.572} C_VEL
LIN {X 0,Y 233.328,Z 1274.251,A -85,B 0,C 180,E1 5293.308,E2 5293.308} C_VEL
LIN {X 0,Y 235.495,Z 1270.462,A -85,B 0,C 180,E1 5288.053,E2 5288.053} C_VEL
LIN {X 0,Y 239.166,Z 1265.353,A -85,B 0,C 180,E1 5282.614,E2 5282.614} C_VEL
LIN {X 0,Y 244.372,Z 1259.053,A -85,B 0,C 180,E1 5277.303,E2 5277.303} C_VEL
LIN {X 0,Y 252.985,Z 1249.643,A -85,B 0,C 180,E1 5271.06,E2 5271.06} C_VEL
LIN {X 0,Y 262.668,Z 1239.452,A -85,B 0,C 180,E1 5265.838,E2 5265.838} C_VEL
LIN {X 0,Y 272.105,Z 1229.703,A -85,B 0,C 180,E1 5261.753,E2 5261.753} C_VEL
LIN {X 0,Y 282.733,Z 1218.683,A -85,B 0,C 180,E1 5257.935,E2 5257.935} C_VEL
LIN {X 0,Y 296.904,Z 1203.7,A -85,B 0,C 180,E1 5253.707,E2 5253.707} C_VEL
LIN {X 0,Y 311.109,Z 1187.766,A -85,B 0,C 180,E1 5250.163,E2 5250.163} C_VEL
LIN {X 0,Y 322.807,Z 1174.057,A -85,B 0,C 180,E1 5247.634,E2 5247.634} C_VEL
LIN {X 0,Y 335.079,Z 1158.902,A -85,B 0,C 180,E1 5245.283,E2 5245.283} C_VEL
LIN {X 0,Y 349.407,Z 1140.079,A -85,B 0,C 180,E1 5242.854,E2 5242.854} C_VEL
LIN {X 0,Y 363.899,Z 1119.126,A -85,B 0,C 180,E1 5240.67,E2 5240.67} C_VEL
LIN {X 0,Y 375.213,Z 1101.386,A -85,B 0,C 180,E1 5239.134,E2 5239.134} C_VEL
LIN {X 0,Y 385.741,Z 1083.469,A -85,B 0,C 180,E1 5237.811,E2 5237.811} C_VEL
LIN {X 0,Y 396.414,Z 1063.591,A -85,B 0,C 180,E1 5236.562,E2 5236.562} C_VEL
LIN {X 0,Y 408.387,Z 1038.647,A -85,B 0,C 180,E1 5235.272,E2 5235.272} C_VEL
LIN {X 0,Y 417.93,Z 1015.695,A -85,B 0,C 180,E1 5234.309,E2 5234.309} C_VEL
LIN {X 0,Y 425.211,Z 995.871,A -85,B 0,C 180,E1 5233.616,E2 5233.616} C_VEL
LIN {X 0,Y 431.806,Z 975.323,A -85,B 0,C 180,E1 5233.016,E2 5233.016} C_VEL
LIN {X 0,Y 437.881,Z 953.136,A -85,B 0,C 180,E1 5232.484,E2 5232.484} C_VEL
LIN {X 0,Y 444.139,Z 924.499,A -85,B 0,C 180,E1 5231.95,E2 5231.95} C_VEL
LIN {X 0,Y 447.983,Z 899.653,A -85,B 0,C 180,E1 5231.556,E2 5231.556} C_VEL
LIN {X 0,Y 468.954,Z 701.207,A -85,B 0,C 180,E1 5228.75,E2 5228.75} C_VEL
LIN {X 0,Y 467.555,Z 698.415,A -85,B 0,C 180,E1 5227.249,E2 5227.249} C_VEL
LIN {X 0,Y 466.082,Z 695.177,A -85,B 0,C 180,E1 5225.17,E2 5225.17} C_VEL
LIN {X 0,Y 464.714,Z 691.299,A -85,B 0,C 180,E1 5221.233,E2 5221.233} C_VEL
LIN {X 0,Y 464.629,Z 691.014,A -85,B 0,C 180,E1 5219.63,E2 5219.63} C_VEL
LIN {X 0,Y 464.708,Z 691.241,A -85,B 0,C 180,E1 5218.644,E2 5218.644} C_VEL
LIN {X 0,Y 466.46,Z 695.967,A -85,B 0,C 180,E1 5214.033,E2 5214.033} C_VEL
LIN {X 0,Y 468.54,Z 700.341,A -85,B 0,C 180,E1 5211.471,E2 5211.471} C_VEL
LIN {X 0,Y 468.891,Z 701.383,A -85,B 0,C 180,E1 5211.084,E2 5211.084} C_VEL
LIN {X 0,Y 448.114,Z 897.77,A -85,B 0,C 180,E1 5208.309,E2 5208.309} C_VEL
LIN {X 0,Y 444.173,Z 923.113,A -85,B 0,C 180,E1 5207.908,E2 5207.908} C_VEL
LIN {X 0,Y 438.065,Z 951.028,A -85,B 0,C 180,E1 5207.367,E2 5207.367} C_VEL
LIN {X 0,Y 432.087,Z 972.955,A -85,B 0,C 180,E1 5206.824,E2 5206.824} C_VEL
LIN {X 0,Y 425.706,Z 992.941,A -85,B 0,C 180,E1 5206.226,E2 5206.226} C_VEL
LIN {X 0,Y 418.01,Z 1013.956,A -85,B 0,C 180,E1 5205.472,E2 5205.472} C_VEL
LIN {X 0,Y 407.942,Z 1038.111,A -85,B 0,C 180,E1 5204.427,E2 5204.427} C_VEL
LIN {X 0,Y 396.42,Z 1061.845,A -85,B 0,C 180,E1 5203.159,E2 5203.159} C_VEL
LIN {X 0,Y 386.013,Z 1081.147,A -85,B 0,C 180,E1 5201.928,E2 5201.928} C_VEL
LIN {X 0,Y 375.36,Z 1099.229,A -85,B 0,C 180,E1 5200.565,E2 5200.565} C_VEL
LIN {X 0,Y 363.329,Z 1117.991,A -85,B 0,C 180,E1 5198.902,E2 5198.902} C_VEL
LIN {X 0,Y 347.783,Z 1140.01,A -85,B 0,C 180,E1 5196.517,E2 5196.517} C_VEL
LIN {X 0,Y 335.401,Z 1156.141,A -85,B 0,C 180,E1 5194.388,E2 5194.388} C_VEL
LIN {X 0,Y 323.551,Z 1170.664,A -85,B 0,C 180,E1 5192.115,E2 5192.115} C_VEL
LIN {X 0,Y 311.208,Z 1185,A -85,B 0,C 180,E1 5189.442,E2 5189.442} C_VEL
LIN {X 0,Y 296.406,Z 1201.358,A -85,B 0,C 180,E1 5185.712,E2 5185.712} C_VEL
LIN {X 0,Y 283.537,Z 1214.787,A -85,B 0,C 180,E1 5181.857,E2 5181.857} C_VEL
LIN {X 0,Y 272.89,Z 1225.652,A -85,B 0,C 180,E1 5178.063,E2 5178.063} C_VEL
LIN {X 0,Y 263.393,Z 1235.25,A -85,B 0,C 180,E1 5174.01,E2 5174.01} C_VEL
LIN {X 0,Y 253.3,Z 1245.667,A -85,B 0,C 180,E1 5168.593,E2 5168.593} C_VEL
LIN {X 0,Y 244.932,Z 1254.497,A -85,B 0,C 180,E1 5162.613,E2 5162.613} C_VEL
LIN {X 0,Y 239.621,Z 1260.659,A -85,B 0,C 180,E1 5157.329,E2 5157.329} C_VEL
LIN {X 0,Y 235.976,Z 1265.439,A -85,B 0,C 180,E1 5152.162,E2 5152.162} C_VEL
LIN {X 0,Y 233.726,Z 1269.015,A -85,B 0,C 180,E1 5147.175,E2 5147.175} C_VEL
LIN {X 0,Y 232.518,Z 1271.665,A -85,B 0,C 180,E1 5142.171,E2 5142.171} C_VEL
LIN {X 0,Y 232.033,Z 1273.409,A -85,B 0,C 180,E1 5137.186,E2 5137.186} C_VEL
LIN {X 0,Y 231.92,Z 1274.218,A -85,B 0,C 180,E1 5132.725,E2 5132.725} C_VEL
LIN {X 0,Y 231.91,Z 1274.319,A -85,B 0,C 180,E1 5128.278,E2 5128.278} C_VEL
LIN {X 0,Y 231.998,Z 1273.646,A -85,B 0,C 180,E1 5123.574,E2 5123.574} C_VEL
LIN {X 0,Y 232.415,Z 1271.949,A -85,B 0,C 180,E1 5118.342,E2 5118.342} C_VEL
LIN {X 0,Y 233.533,Z 1269.414,A -85,B 0,C 180,E1 5113.338,E2 5113.338} C_VEL
LIN {X 0,Y 235.791,Z 1265.75,A -85,B 0,C 180,E1 5108.097,E2 5108.097} C_VEL
LIN {X 0,Y 239.43,Z 1260.93,A -85,B 0,C 180,E1 5102.813,E2 5102.813} C_VEL
LIN {X 0,Y 244.552,Z 1254.953,A -85,B 0,C 180,E1 5097.624,E2 5097.624} C_VEL
LIN {X 0,Y 252.085,Z 1246.944,A -85,B 0,C 180,E1 5092.073,E2 5092.073} C_VEL
LIN {X 0,Y 262.796,Z 1235.929,A -85,B 0,C 180,E1 5086.185,E2 5086.185} C_VEL
LIN {X 0,Y 272.725,Z 1225.898,A -85,B 0,C 180,E1 5081.917,E2 5081.917} C_VEL
LIN {X 0,Y 283.361,Z 1215.06,A -85,B 0,C 180,E1 5078.117,E2 5078.117} C_VEL
LIN {X 0,Y 296.895,Z 1200.969,A -85,B 0,C 180,E1 5074.071,E2 5074.071} C_VEL
LIN {X 0,Y 311.018,Z 1185.365,A -85,B 0,C 180,E1 5070.519,E2 5070.519} C_VEL
LIN {X 0,Y 323.426,Z 1170.979,A -85,B 0,C 180,E1 5067.829,E2 5067.829} C_VEL
LIN {X 0,Y 335.969,Z 1155.614,A -85,B 0,C 180,E1 5065.428,E2 5065.428} C_VEL
LIN {X 0,Y 350.039,Z 1137.24,A -85,B 0,C 180,E1 5063.038,E2 5063.038} C_VEL
LIN {X 0,Y 364.719,Z 1116.118,A -85,B 0,C 180,E1 5060.814,E2 5060.814} C_VEL
LIN {X 0,Y 375.985,Z 1098.501,A -85,B 0,C 180,E1 5059.272,E2 5059.272} C_VEL
LIN {X 0,Y 386.538,Z 1080.551,A -85,B 0,C 180,E1 5057.928,E2 5057.928} C_VEL
LIN {X 0,Y 397.128,Z 1060.85,A -85,B 0,C 180,E1 5056.68,E2 5056.68} C_VEL
LIN {X 0,Y 409.474,Z 1034.964,A -85,B 0,C 180,E1 5055.328,E2 5055.328} C_VEL
LIN {X 0,Y 418.401,Z 1013.452,A -85,B 0,C 180,E1 5054.41,E2 5054.41} C_VEL
LIN {X 0,Y 425.758,Z 993.379,A -85,B 0,C 180,E1 5053.691,E2 5053.691} C_VEL
LIN {X 0,Y 432.335,Z 972.815,A -85,B 0,C 180,E1 5053.076,E2 5053.076} C_VEL
LIN {X 0,Y 438.43,Z 950.408,A -85,B 0,C 180,E1 5052.522,E2 5052.522} C_VEL
LIN {X 0,Y 444.736,Z 921.034,A -85,B 0,C 180,E1 5051.961,E2 5051.961} C_VEL
LIN {X 0,Y 448.397,Z 897.202,A -85,B 0,C 180,E1 5051.586,E2 5051.586} C_VEL
LIN {X 0,Y 450.668,Z 877.469,A -85,B 0,C 180,E1 5051.298,E2 5051.298} C_VEL
LIN {X 0,Y 451.253,Z 869.943,A -85,B 0,C 180,E1 5051.067,E2 5051.067} C_VEL
LIN {X 0,Y 452.153,Z 850.411,A -85,B 0,C 180,E1 5050.013,E2 5050.013} C_VEL
LIN {X 0,Y 452.701,Z 843.94,A -85,B 0,C 180,E1 5049.825,E2 5049.825} C_VEL
LIN {X 0,Y 467.287,Z 707.594,A -85,B 0,C 180,E1 5047.933,E2 5047.933} C_VEL
LIN {X 0,Y 465.191,Z 703.161,A -85,B 0,C 180,E1 5045.056,E2 5045.056} C_VEL
LIN {X 0,Y 463.953,Z 699.32,A -85,B 0,C 180,E1 5040.988,E2 5040.988} C_VEL
LIN {X 0,Y 463.957,Z 699.048,A -85,B 0,C 180,E1 5039.383,E2 5039.383} C_VEL
LIN {X 0,Y 465.105,Z 703.08,A -85,B 0,C 180,E1 5035.19,E2 5035.19} C_VEL
LIN {X 0,Y 465.809,Z 704.695,A -85,B 0,C 180,E1 5034.024,E2 5034.024} C_VEL
LIN {X 0,Y 467.311,Z 707.751,A -85,B 0,C 180,E1 5032.137,E2 5032.137} C_VEL
LIN {X 0,Y 446.643,Z 899.688,A -85,B 0,C 180,E1 5029.458,E2 5029.458} C_VEL
LIN {X 0,Y 442.62,Z 925.21,A -85,B 0,C 180,E1 5029.061,E2 5029.061} C_VEL
LIN {X 0,Y 436.351,Z 953.319,A -85,B 0,C 180,E1 5028.549,E2 5028.549} C_VEL
LIN {X 0,Y 430.248,Z 975.299,A -85,B 0,C 180,E1 5028.037,E2 5028.037} C_VEL
LIN {X 0,Y 423.618,Z 995.685,A -85,B 0,C 180,E1 5027.458,E2 5027.458} C_VEL
LIN {X 0,Y 415.965,Z 1016.206,A -85,B 0,C 180,E1 5026.759,E2 5026.759} C_VEL
LIN {X 0,Y 405.414,Z 1041.065,A -85,B 0,C 180,E1 5025.732,E2 5025.732} C_VEL
LIN {X 0,Y 393.74,Z 1064.66,A -85,B 0,C 180,E1 5024.522,E2 5024.522} C_VEL
LIN {X 0,Y 383.464,Z 1083.446,A -85,B 0,C 180,E1 5023.364,E2 5023.364} C_VEL
LIN {X 0,Y 372.965,Z 1100.988,A -85,B 0,C 180,E1 5022.102,E2 5022.102} C_VEL
LIN {X 0,Y 361.033,Z 1119.341,A -85,B 0,C 180,E1 5020.544,E2 5020.544} C_VEL
LIN {X 0,Y 345.174,Z 1141.608,A -85,B 0,C 180,E1 5018.236,E2 5018.236} C_VEL
LIN {X 0,Y 331.576,Z 1159.029,A -85,B 0,C 180,E1 5016.006,E2 5016.006} C_VEL
LIN {X 0,Y 318.991,Z 1174.162,A -85,B 0,C 180,E1 5013.682,E2 5013.682} C_VEL
LIN {X 0,Y 306.27,Z 1188.624,A -85,B 0,C 180,E1 5011.023,E2 5011.023} C_VEL
LIN {X 0,Y 291.018,Z 1205.063,A -85,B 0,C 180,E1 5007.314,E2 5007.314} C_VEL
LIN {X 0,Y 277.609,Z 1218.707,A -85,B 0,C 180,E1 5003.423,E2 5003.423} C_VEL
LIN {X 0,Y 266.541,Z 1229.711,A -85,B 0,C 180,E1 4999.586,E2 4999.586} C_VEL
LIN {X 0,Y 256.215,Z 1239.912,A -85,B 0,C 180,E1 4995.244,E2 4995.244} C_VEL
LIN {X 0,Y 245.352,Z 1250.785,A -85,B 0,C 180,E1 4989.465,E2 4989.465} C_VEL
LIN {X 0,Y 237.071,Z 1259.327,A -85,B 0,C 180,E1 4983.53,E2 4983.53} C_VEL
LIN {X 0,Y 231.797,Z 1265.309,A -85,B 0,C 180,E1 4978.317,E2 4978.317} C_VEL
LIN {X 0,Y 227.963,Z 1270.243,A -85,B 0,C 180,E1 4972.912,E2 4972.912} C_VEL
LIN {X 0,Y 225.573,Z 1274.028,A -85,B 0,C 180,E1 4967.534,E2 4967.534} C_VEL
LIN {X 0,Y 224.393,Z 1276.705,A -85,B 0,C 180,E1 4962.342,E2 4962.342} C_VEL
LIN {X 0,Y 223.977,Z 1278.452,A -85,B 0,C 180,E1 4957.173,E2 4957.173} C_VEL
LIN {X 0,Y 223.914,Z 1279.207,A -85,B 0,C 180,E1 4952.808,E2 4952.808} C_VEL
LIN {X 0,Y 223.906,Z 1279.319,A -85,B 0,C 180,E1 4948.457,E2 4948.457} C_VEL
LIN {X 0,Y 223.954,Z 1278.647,A -85,B 0,C 180,E1 4943.584,E2 4943.584} C_VEL
LIN {X 0,Y 224.358,Z 1276.799,A -85,B 0,C 180,E1 4937.902,E2 4937.902} C_VEL
LIN {X 0,Y 225.491,Z 1274.161,A -85,B 0,C 180,E1 4932.71,E2 4932.71} C_VEL
LIN {X 0,Y 227.855,Z 1270.371,A -85,B 0,C 180,E1 4927.277,E2 4927.277} C_VEL
LIN {X 0,Y 231.595,Z 1265.519,A -85,B 0,C 180,E1 4921.92,E2 4921.92} C_VEL
LIN {X 0,Y 236.798,Z 1259.574,A -85,B 0,C 180,E1 4916.7,E2 4916.7} C_VEL
LIN {X 0,Y 244.628,Z 1251.426,A -85,B 0,C 180,E1 4910.984,E2 4910.984} C_VEL
LIN {X 0,Y 255.777,Z 1240.283,A -85,B 0,C 180,E1 4904.956,E2 4904.956} C_VEL
LIN {X 0,Y 266.043,Z 1230.128,A -85,B 0,C 180,E1 4900.601,E2 4900.601} C_VEL
LIN {X 0,Y 276.719,Z 1219.503,A -85,B 0,C 180,E1 4896.857,E2 4896.857} C_VEL
LIN {X 0,Y 288.509,Z 1207.481,A -85,B 0,C 180,E1 4893.353,E2 4893.353} C_VEL
LIN {X 0,Y 304.238,Z 1190.77,A -85,B 0,C 180,E1 4889.427,E2 4889.427} C_VEL
LIN {X 0,Y 318.294,Z 1174.812,A -85,B 0,C 180,E1 4886.447,E2 4886.447} C_VEL
LIN {X 0,Y 330.851,Z 1159.738,A -85,B 0,C 180,E1 4884.113,E2 4884.113} C_VEL
LIN {X 0,Y 343.52,Z 1143.547,A -85,B 0,C 180,E1 4882.013,E2 4882.013} C_VEL
LIN {X 0,Y 358.64,Z 1122.695,A -85,B 0,C 180,E1 4879.782,E2 4879.782} C_VEL
LIN {X 0,Y 372.169,Z 1101.978,A -85,B 0,C 180,E1 4877.991,E2 4877.991} C_VEL
LIN {X 0,Y 382.87,Z 1084.144,A -85,B 0,C 180,E1 4876.695,E2 4876.695} C_VEL
LIN {X 0,Y 393.3,Z 1065.123,A -85,B 0,C 180,E1 4875.515,E2 4875.515} C_VEL
LIN {X 0,Y 404.573,Z 1042.398,A -85,B 0,C 180,E1 4874.341,E2 4874.341} C_VEL
LIN {X 0,Y 415.115,Z 1017.864,A -85,B 0,C 180,E1 4873.31,E2 4873.31} C_VEL
LIN {X 0,Y 423.115,Z 996.537,A -85,B 0,C 180,E1 4872.576,E2 4872.576} C_VEL
LIN {X 0,Y 429.835,Z 975.967,A -85,B 0,C 180,E1 4871.987,E2 4871.987} C_VEL
LIN {X 0,Y 435.874,Z 954.331,A -85,B 0,C 180,E1 4871.479,E2 4871.479} C_VEL
LIN {X 0,Y 442.048,Z 927.276,A -85,B 0,C 180,E1 4870.978,E2 4870.978} C_VEL
LIN {X 0,Y 446.364,Z 900.161,A -85,B 0,C 180,E1 4870.554,E2 4870.554} C_VEL
LIN {X 0,Y 461.643,Z 758.2,A -85,B 0,C 180,E1 4868.565,E2 4868.565} C_VEL
LIN {X 0,Y 467.087,Z 707.445,A -85,B 0,C 180,E1 4867.844,E2 4867.844} C_VEL
LIN {X 0,Y 465.027,Z 703.057,A -85,B 0,C 180,E1 4865.058,E2 4865.058} C_VEL
LIN {X 0,Y 463.725,Z 699.179,A -85,B 0,C 180,E1 4861.112,E2 4861.112} C_VEL
LIN {X 0,Y 463.719,Z 699.122,A -85,B 0,C 180,E1 4858.764,E2 4858.764} C_VEL
LIN {X 0,Y 465.356,Z 703.77,A -85,B 0,C 180,E1 4854.204,E2 4854.204} C_VEL
LIN {X 0,Y 467.06,Z 707.526,A -85,B 0,C 180,E1 4851.972,E2 4851.972} C_VEL
LIN {X 0,Y 446.548,Z 897.955,A -85,B 0,C 180,E1 4849.316,E2 4849.316} C_VEL
LIN {X 0,Y 442.487,Z 923.656,A -85,B 0,C 180,E1 4848.917,E2 4848.917} C_VEL
LIN {X 0,Y 436.329,Z 951.318,A -85,B 0,C 180,E1 4848.392,E2 4848.392} C_VEL
LIN {X 0,Y 430.324,Z 973.053,A -85,B 0,C 180,E1 4847.867,E2 4847.867} C_VEL
LIN {X 0,Y 423.857,Z 993.038,A -85,B 0,C 180,E1 4847.285,E2 4847.285} C_VEL
LIN {X 0,Y 416.336,Z 1013.331,A -85,B 0,C 180,E1 4846.578,E2 4846.578} C_VEL
LIN {X 0,Y 406.705,Z 1036.202,A -85,B 0,C 180,E1 4845.622,E2 4845.622} C_VEL
LIN {X 0,Y 394.606,Z 1061.05,A -85,B 0,C 180,E1 4844.345,E2 4844.345} C_VEL
LIN {X 0,Y 383.98,Z 1080.509,A -85,B 0,C 180,E1 4843.138,E2 4843.138} C_VEL
LIN {X 0,Y 373.539,Z 1097.992,A -85,B 0,C 180,E1 4841.859,E2 4841.859} C_VEL
LIN {X 0,Y 362.282,Z 1115.321,A -85,B 0,C 180,E1 4840.383,E2 4840.383} C_VEL
LIN {X 0,Y 347.698,Z 1136.053,A -85,B 0,C 180,E1 4838.264,E2 4838.264} C_VEL
LIN {X 0,Y 333.052,Z 1154.821,A -85,B 0,C 180,E1 4835.883,E2 4835.883} C_VEL
LIN {X 0,Y 320.467,Z 1169.917,A -85,B 0,C 180,E1 4833.575,E2 4833.575} C_VEL
LIN {X 0,Y 308.431,Z 1183.562,A -85,B 0,C 180,E1 4831.087,E2 4831.087} C_VEL
LIN {X 0,Y 295.686,Z 1197.298,A -85,B 0,C 180,E1 4828.085,E2 4828.085} C_VEL
LIN {X 0,Y 280.186,Z 1213.174,A -85,B 0,C 180,E1 4823.763,E2 4823.763} C_VEL
LIN {X 0,Y 268.404,Z 1224.725,A -85,B 0,C 180,E1 4819.797,E2 4819.797} C_VEL
LIN {X 0,Y 258.384,Z 1234.434,A -85,B 0,C 180,E1 4815.724,E2 4815.724} C_VEL
LIN {X 0,Y 249.168,Z 1243.353,A -85,B 0,C 180,E1 4811.163,E2 4811.163} C_VEL
LIN {X 0,Y 239.805,Z 1252.788,A -85,B 0,C 180,E1 4805.134,E2 4805.134} C_VEL
LIN {X 0,Y 232.735,Z 1260.248,A -85,B 0,C 180,E1 4798.769,E2 4798.769} C_VEL
LIN {X 0,Y 228.518,Z 1265.326,A -85,B 0,C 180,E1 4793.198,E2 4793.198} C_VEL
LIN {X 0,Y 225.985,Z 1269.002,A -85,B 0,C 180,E1 4787.957,E2 4787.957} C_VEL
LIN {X 0,Y 224.631,Z 1271.642,A -85,B 0,C 180,E1 4782.866,E2 4782.866} C_VEL
LIN {X 0,Y 224.048,Z 1273.431,A -85,B 0,C 180,E1 4777.701,E2 4777.701} C_VEL
LIN {X 0,Y 223.924,Z 1274.283,A -85,B 0,C 180,E1 4773.079,E2 4773.079} C_VEL
LIN {X 0,Y 223.905,Z 1274.429,A -85,B 0,C 180,E1 4768.472,E2 4768.472} C_VEL
LIN {X 0,Y 224.008,Z 1273.734,A -85,B 0,C 180,E1 4763.343,E2 4763.343} C_VEL
LIN {X 0,Y 224.48,Z 1272.038,A -85,B 0,C 180,E1 4757.924,E2 4757.924} C_VEL
LIN {X 0,Y 225.704,Z 1269.503,A -85,B 0,C 180,E1 4752.742,E2 4752.742} C_VEL
LIN {X 0,Y 228.162,Z 1265.84,A -85,B 0,C 180,E1 4747.325,E2 4747.325} C_VEL
LIN {X 0,Y 231.991,Z 1261.131,A -85,B 0,C 180,E1 4741.989,E2 4741.989} C_VEL
LIN {X 0,Y 237.557,Z 1255.043,A -85,B 0,C 180,E1 4736.548,E2 4736.548} C_VEL
LIN {X 0,Y 245.922,Z 1246.685,A -85,B 0,C 180,E1 4730.645,E2 4730.645} C_VEL
LIN {X 0,Y 256.82,Z 1236.019,A -85,B 0,C 180,E1 4724.892,E2 4724.892} C_VEL
LIN {X 0,Y 267.187,Z 1225.988,A -85,B 0,C 180,E1 4720.577,E2 4720.577} C_VEL
LIN {X 0,Y 278.258,Z 1215.15,A -85,B 0,C 180,E1 4716.757,E2 4716.757} C_VEL
LIN {X 0,Y 292.287,Z 1201.059,A -85,B 0,C 180,E1 4712.711,E2 4712.711} C_VEL
LIN {X 0,Y 306.864,Z 1185.453,A -85,B 0,C 180,E1 4709.177,E2 4709.177} C_VEL
LIN {X 0,Y 319.554,Z 1171.147,A -85,B 0,C 180,E1 4706.522,E2 4706.522} C_VEL
LIN {X 0,Y 332.417,Z 1155.788,A -85,B 0,C 180,E1 4704.147,E2 4704.147} C_VEL
LIN {X 0,Y 347.511,Z 1136.521,A -85,B 0,C 180,E1 4701.684,E2 4701.684} C_VEL
LIN {X 0,Y 361.872,Z 1116.204,A -85,B 0,C 180,E1 4699.594,E2 4699.594} C_VEL
LIN {X 0,Y 373.357,Z 1098.586,A -85,B 0,C 180,E1 4698.084,E2 4698.084} C_VEL
LIN {X 0,Y 383.721,Z 1081.294,A -85,B 0,C 180,E1 4696.813,E2 4696.813} C_VEL
LIN {X 0,Y 394.002,Z 1062.564,A -85,B 0,C 180,E1 4695.642,E2 4695.642} C_VEL
LIN {X 0,Y 405.666,Z 1039.012,A -85,B 0,C 180,E1 4694.407,E2 4694.407} C_VEL
LIN {X 0,Y 416.169,Z 1014.281,A -85,B 0,C 180,E1 4693.36,E2 4693.36} C_VEL
LIN {X 0,Y 423.692,Z 994.117,A -85,B 0,C 180,E1 4692.652,E2 4692.652} C_VEL
LIN {X 0,Y 430.386,Z 973.548,A -85,B 0,C 180,E1 4692.049,E2 4692.049} C_VEL
LIN {X 0,Y 436.331,Z 952.128,A -85,B 0,C 180,E1 4691.529,E2 4691.529} C_VEL
LIN {X 0,Y 442.424,Z 925.274,A -85,B 0,C 180,E1 4691.013,E2 4691.013} C_VEL
LIN {X 0,Y 446.713,Z 898.377,A -85,B 0,C 180,E1 4690.594,E2 4690.594} C_VEL
LIN {X 0,Y 452.701,Z 843.94,A -85,B 0,C 180,E1 4689.825,E2 4689.825} C_VEL
LIN {X 0,Y 453.322,Z 836.42,A -85,B 0,C 180,E1 4689.59,E2 4689.59} C_VEL
LIN {X 0,Y 454.429,Z 816.903,A -85,B 0,C 180,E1 4688.54,E2 4688.54} C_VEL
LIN {X 0,Y 455.02,Z 810.431,A -85,B 0,C 180,E1 4688.359,E2 4688.359} C_VEL
LIN {X 0,Y 465.51,Z 714.226,A -85,B 0,C 180,E1 4687.033,E2 4687.033} C_VEL
LIN {X 0,Y 464.141,Z 711.042,A -85,B 0,C 180,E1 4684.943,E2 4684.943} C_VEL
LIN {X 0,Y 462.971,Z 707.199,A -85,B 0,C 180,E1 4680.866,E2 4680.866} C_VEL
LIN {X 0,Y 462.971,Z 707.181,A -85,B 0,C 180,E1 4679.258,E2 4679.258} C_VEL
LIN {X 0,Y 464.129,Z 711.059,A -85,B 0,C 180,E1 4675.18,E2 4675.18} C_VEL
LIN {X 0,Y 465.528,Z 714.503,A -85,B 0,C 180,E1 4673.024,E2 4673.024} C_VEL
LIN {X 0,Y 445.242,Z 899.621,A -85,B 0,C 180,E1 4670.475,E2 4670.475} C_VEL
LIN {X 0,Y 441.171,Z 925.108,A -85,B 0,C 180,E1 4670.086,E2 4670.086} C_VEL
LIN {X 0,Y 434.819,Z 953.264,A -85,B 0,C 180,E1 4669.588,E2 4669.588} C_VEL
LIN {X 0,Y 428.648,Z 975.22,A -85,B 0,C 180,E1 4669.093,E2 4669.093} C_VEL
LIN {X 0,Y 422.01,Z 995.391,A -85,B 0,C 180,E1 4668.537,E2 4668.537} C_VEL
LIN {X 0,Y 414.183,Z 1016.125,A -85,B 0,C 180,E1 4667.851,E2 4667.851} C_VEL
LIN {X 0,Y 403.485,Z 1040.982,A -85,B 0,C 180,E1 4666.853,E2 4666.853} C_VEL
LIN {X 0,Y 392.031,Z 1063.844,A -85,B 0,C 180,E1 4665.715,E2 4665.715} C_VEL
LIN {X 0,Y 381.629,Z 1082.624,A -85,B 0,C 180,E1 4664.592,E2 4664.592} C_VEL
LIN {X 0,Y 370.939,Z 1100.232,A -85,B 0,C 180,E1 4663.365,E2 4663.365} C_VEL
LIN {X 0,Y 359.257,Z 1117.943,A -85,B 0,C 180,E1 4661.906,E2 4661.906} C_VEL
LIN {X 0,Y 344.582,Z 1138.456,A -85,B 0,C 180,E1 4659.876,E2 4659.876} C_VEL
LIN {X 0,Y 329.056,Z 1158.011,A -85,B 0,C 180,E1 4657.461,E2 4657.461} C_VEL
LIN {X 0,Y 316.128,Z 1173.224,A -85,B 0,C 180,E1 4655.179,E2 4655.179} C_VEL
LIN {X 0,Y 303.726,Z 1186.986,A -85,B 0,C 180,E1 4652.713,E2 4652.713} C_VEL
LIN {X 0,Y 290.565,Z 1200.853,A -85,B 0,C 180,E1 4649.723,E2 4649.723} C_VEL
LIN {X 0,Y 273.892,Z 1217.463,A -85,B 0,C 180,E1 4645.211,E2 4645.211} C_VEL
LIN {X 0,Y 261.744,Z 1229.065,A -85,B 0,C 180,E1 4641.208,E2 4641.208} C_VEL
LIN {X 0,Y 251.318,Z 1238.895,A -85,B 0,C 180,E1 4637.047,E2 4637.047} C_VEL
LIN {X 0,Y 241.347,Z 1248.332,A -85,B 0,C 180,E1 4632.133,E2 4632.133} C_VEL
LIN {X 0,Y 231.08,Z 1258.317,A -85,B 0,C 180,E1 4625.427,E2 4625.427} C_VEL
LIN {X 0,Y 224.725,Z 1264.962,A -85,B 0,C 180,E1 4619.586,E2 4619.586} C_VEL
LIN {X 0,Y 220.568,Z 1269.9,A -85,B 0,C 180,E1 4614.069,E2 4614.069} C_VEL
LIN {X 0,Y 217.976,Z 1273.615,A -85,B 0,C 180,E1 4608.721,E2 4608.721} C_VEL
LIN {X 0,Y 216.544,Z 1276.385,A -85,B 0,C 180,E1 4603.34,E2 4603.34} C_VEL
LIN {X 0,Y 215.996,Z 1278.155,A -85,B 0,C 180,E1 4598.243,E2 4598.243} C_VEL
LIN {X 0,Y 215.915,Z 1279.05,A -85,B 0,C 180,E1 4593.709,E2 4593.709} C_VEL
LIN {X 0,Y 215.899,Z 1279.254,A -85,B 0,C 180,E1 4588.666,E2 4588.666} C_VEL
LIN {X 0,Y 215.953,Z 1278.628,A -85,B 0,C 180,E1 4583.613,E2 4583.613} C_VEL
LIN {X 0,Y 216.378,Z 1276.825,A -85,B 0,C 180,E1 4577.72,E2 4577.72} C_VEL
LIN {X 0,Y 217.737,Z 1273.977,A -85,B 0,C 180,E1 4571.914,E2 4571.914} C_VEL
LIN {X 0,Y 220.256,Z 1270.28,A -85,B 0,C 180,E1 4566.447,E2 4566.447} C_VEL
LIN {X 0,Y 224.297,Z 1265.406,A -85,B 0,C 180,E1 4560.897,E2 4560.897} C_VEL
LIN {X 0,Y 229.852,Z 1259.481,A -85,B 0,C 180,E1 4555.555,E2 4555.555} C_VEL
LIN {X 0,Y 238.156,Z 1251.333,A -85,B 0,C 180,E1 4549.71,E2 4549.71} C_VEL
LIN {X 0,Y 249.9,Z 1240.19,A -85,B 0,C 180,E1 4543.59,E2 4543.59} C_VEL
LIN {X 0,Y 260.635,Z 1230.034,A -85,B 0,C 180,E1 4539.193,E2 4539.193} C_VEL
LIN {X 0,Y 271.499,Z 1219.65,A -85,B 0,C 180,E1 4535.514,E2 4535.514} C_VEL
LIN {X 0,Y 283.972,Z 1207.387,A -85,B 0,C 180,E1 4531.936,E2 4531.936} C_VEL
LIN {X 0,Y 300.212,Z 1190.676,A -85,B 0,C 180,E1 4528.034,E2 4528.034} C_VEL
LIN {X 0,Y 314.664,Z 1174.718,A -85,B 0,C 180,E1 4525.086,E2 4525.086} C_VEL
LIN {X 0,Y 327.535,Z 1159.644,A -85,B 0,C 180,E1 4522.783,E2 4522.783} C_VEL
LIN {X 0,Y 340.333,Z 1143.657,A -85,B 0,C 180,E1 4520.74,E2 4520.74} C_VEL
LIN {X 0,Y 355.515,Z 1123.212,A -85,B 0,C 180,E1 4518.585,E2 4518.585} C_VEL
LIN {X 0,Y 369.109,Z 1102.833,A -85,B 0,C 180,E1 4516.849,E2 4516.849} C_VEL
LIN {X 0,Y 380.146,Z 1084.819,A -85,B 0,C 180,E1 4515.563,E2 4515.563} C_VEL
LIN {X 0,Y 390.756,Z 1065.842,A -85,B 0,C 180,E1 4514.407,E2 4514.407} C_VEL
LIN {X 0,Y 401.197,Z 1045.224,A -85,B 0,C 180,E1 4513.355,E2 4513.355} C_VEL
LIN {X 0,Y 413.018,Z 1018.541,A -85,B 0,C 180,E1 4512.244,E2 4512.244} C_VEL
LIN {X 0,Y 421.427,Z 996.441,A -85,B 0,C 180,E1 4511.503,E2 4511.503} C_VEL
LIN {X 0,Y 428.231,Z 975.869,A -85,B 0,C 180,E1 4510.931,E2 4510.931} C_VEL
LIN {X 0,Y 434.451,Z 953.823,A -85,B 0,C 180,E1 4510.43,E2 4510.43} C_VEL
LIN {X 0,Y 440.716,Z 926.443,A -85,B 0,C 180,E1 4509.94,E2 4509.94} C_VEL
LIN {X 0,Y 444.977,Z 899.93,A -85,B 0,C 180,E1 4509.535,E2 4509.535} C_VEL
LIN {X 0,Y 462.321,Z 741.551,A -85,B 0,C 180,E1 4507.35,E2 4507.35} C_VEL
LIN {X 0,Y 465.329,Z 714.105,A -85,B 0,C 180,E1 4506.973,E2 4506.973} C_VEL
LIN {X 0,Y 463.9,Z 710.835,A -85,B 0,C 180,E1 4504.822,E2 4504.822} C_VEL
LIN {X 0,Y 462.737,Z 707.06,A -85,B 0,C 180,E1 4500.99,E2 4500.99} C_VEL
LIN {X 0,Y 462.733,Z 707.002,A -85,B 0,C 180,E1 4498.886,E2 4498.886} C_VEL
LIN {X 0,Y 464.291,Z 711.681,A -85,B 0,C 180,E1 4494.315,E2 4494.315} C_VEL
LIN {X 0,Y 465.285,Z 714.199,A -85,B 0,C 180,E1 4492.86,E2 4492.86} C_VEL
LIN {X 0,Y 445.121,Z 898.141,A -85,B 0,C 180,E1 4490.329,E2 4490.329} C_VEL
LIN {X 0,Y 440.922,Z 924.295,A -85,B 0,C 180,E1 4489.931,E2 4489.931} C_VEL
LIN {X 0,Y 434.719,Z 951.661,A -85,B 0,C 180,E1 4489.425,E2 4489.425} C_VEL
LIN {X 0,Y 428.704,Z 973.15,A -85,B 0,C 180,E1 4488.919,E2 4488.919} C_VEL
LIN {X 0,Y 422.155,Z 993.134,A -85,B 0,C 180,E1 4488.353,E2 4488.353} C_VEL
LIN {X 0,Y 414.533,Z 1013.426,A -85,B 0,C 180,E1 4487.666,E2 4487.666} C_VEL
LIN {X 0,Y 404.533,Z 1036.831,A -85,B 0,C 180,E1 4486.711,E2 4486.711} C_VEL
LIN {X 0,Y 392.485,Z 1061.145,A -85,B 0,C 180,E1 4485.491,E2 4485.491} C_VEL
LIN {X 0,Y 381.691,Z 1080.603,A -85,B 0,C 180,E1 4484.311,E2 4484.311} C_VEL
LIN {X 0,Y 371.068,Z 1098.086,A -85,B 0,C 180,E1 4483.063,E2 4483.063} C_VEL
LIN {X 0,Y 359.371,Z 1115.755,A -85,B 0,C 180,E1 4481.588,E2 4481.588} C_VEL
LIN {X 0,Y 344.515,Z 1136.421,A -85,B 0,C 180,E1 4479.509,E2 4479.509} C_VEL
LIN {X 0,Y 329.36,Z 1155.38,A -85,B 0,C 180,E1 4477.133,E2 4477.133} C_VEL
LIN {X 0,Y 316.856,Z 1170.011,A -85,B 0,C 180,E1 4474.921,E2 4474.921} C_VEL
LIN {X 0,Y 304.125,Z 1184.05,A -85,B 0,C 180,E1 4472.382,E2 4472.382} C_VEL
LIN {X 0,Y 290.02,Z 1198.784,A -85,B 0,C 180,E1 4469.151,E2 4469.151} C_VEL
LIN {X 0,Y 274.085,Z 1214.417,A -85,B 0,C 180,E1 4464.802,E2 4464.802} C_VEL
LIN {X 0,Y 262.515,Z 1225.329,A -85,B 0,C 180,E1 4460.994,E2 4460.994} C_VEL
LIN {X 0,Y 252.111,Z 1234.981,A -85,B 0,C 180,E1 4456.873,E2 4456.873} C_VEL
LIN {X 0,Y 241.967,Z 1244.36,A -85,B 0,C 180,E1 4451.942,E2 4451.942} C_VEL
LIN {X 0,Y 231.388,Z 1254.382,A -85,B 0,C 180,E1 4445.087,E2 4445.087} C_VEL
LIN {X 0,Y 225.246,Z 1260.591,A -85,B 0,C 180,E1 4439.528,E2 4439.528} C_VEL
LIN {X 0,Y 220.793,Z 1265.621,A -85,B 0,C 180,E1 4433.776,E2 4433.776} C_VEL
LIN {X 0,Y 218.039,Z 1269.352,A -85,B 0,C 180,E1 4428.177,E2 4428.177} C_VEL
LIN {X 0,Y 216.617,Z 1271.955,A -85,B 0,C 180,E1 4422.808,E2 4422.808} C_VEL
LIN {X 0,Y 216.046,Z 1273.653,A -85,B 0,C 180,E1 4417.453,E2 4417.453} C_VEL
LIN {X 0,Y 215.92,Z 1274.415,A -85,B 0,C 180,E1 4412.662,E2 4412.662} C_VEL
LIN {X 0,Y 215.912,Z 1274.494,A -85,B 0,C 180,E1 4408.15,E2 4408.15} C_VEL
LIN {X 0,Y 216.019,Z 1273.822,A -85,B 0,C 180,E1 4403.096,E2 4403.096} C_VEL
LIN {X 0,Y 216.55,Z 1272.126,A -85,B 0,C 180,E1 4397.475,E2 4397.475} C_VEL
LIN {X 0,Y 218,Z 1269.435,A -85,B 0,C 180,E1 4391.836,E2 4391.836} C_VEL
LIN {X 0,Y 220.769,Z 1265.691,A -85,B 0,C 180,E1 4386.19,E2 4386.19} C_VEL
LIN {X 0,Y 225.119,Z 1260.764,A -85,B 0,C 180,E1 4380.524,E2 4380.524} C_VEL
LIN {X 0,Y 231.597,Z 1254.235,A -85,B 0,C 180,E1 4374.664,E2 4374.664} C_VEL
LIN {X 0,Y 241.945,Z 1244.448,A -85,B 0,C 180,E1 4367.983,E2 4367.983} C_VEL
LIN {X 0,Y 251.953,Z 1235.199,A -85,B 0,C 180,E1 4363.108,E2 4363.108} C_VEL
LIN {X 0,Y 262.427,Z 1225.496,A -85,B 0,C 180,E1 4358.953,E2 4358.953} C_VEL
LIN {X 0,Y 274.529,Z 1214.101,A -85,B 0,C 180,E1 4354.98,E2 4354.98} C_VEL
LIN {X 0,Y 291.176,Z 1197.715,A -85,B 0,C 180,E1 4350.482,E2 4350.482} C_VEL
LIN {X 0,Y 304.306,Z 1184.009,A -85,B 0,C 180,E1 4347.498,E2 4347.498} C_VEL
LIN {X 0,Y 316.685,Z 1170.378,A -85,B 0,C 180,E1 4345.03,E2 4345.03} C_VEL
LIN {X 0,Y 330.341,Z 1154.407,A -85,B 0,C 180,E1 4342.623,E2 4342.623} C_VEL
LIN {X 0,Y 346.947,Z 1133.325,A -85,B 0,C 180,E1 4340.05,E2 4340.05} C_VEL
LIN {X 0,Y 360.232,Z 1114.764,A -85,B 0,C 180,E1 4338.218,E2 4338.218} C_VEL
LIN {X 0,Y 371.735,Z 1097.341,A -85,B 0,C 180,E1 4336.776,E2 4336.776} C_VEL
LIN {X 0,Y 382.378,Z 1079.777,A -85,B 0,C 180,E1 4335.533,E2 4335.533} C_VEL
LIN {X 0,Y 394.939,Z 1056.982,A -85,B 0,C 180,E1 4334.177,E2 4334.177} C_VEL
LIN {X 0,Y 406.368,Z 1033.124,A -85,B 0,C 180,E1 4333.028,E2 4333.028} C_VEL
LIN {X 0,Y 414.776,Z 1013.347,A -85,B 0,C 180,E1 4332.234,E2 4332.234} C_VEL
LIN {X 0,Y 422.449,Z 992.914,A -85,B 0,C 180,E1 4331.543,E2 4331.543} C_VEL
LIN {X 0,Y 429.231,Z 972.149,A -85,B 0,C 180,E1 4330.959,E2 4330.959} C_VEL
LIN {X 0,Y 435.966,Z 947.764,A -85,B 0,C 180,E1 4330.396,E2 4330.396} C_VEL
LIN {X 0,Y 441.946,Z 919.704,A -85,B 0,C 180,E1 4329.901,E2 4329.901} C_VEL
LIN {X 0,Y 445.531,Z 896.711,A -85,B 0,C 180,E1 4329.554,E2 4329.554} C_VEL
LIN {X 0,Y 455.02,Z 810.431,A -85,B 0,C 180,E1 4328.359,E2 4328.359} C_VEL
LIN {X 0,Y 455.695,Z 802.906,A -85,B 0,C 180,E1 4328.132,E2 4328.132} C_VEL
LIN {X 0,Y 457.007,Z 783.397,A -85,B 0,C 180,E1 4327.087,E2 4327.087} C_VEL
LIN {X 0,Y 457.629,Z 776.927,A -85,B 0,C 180,E1 4326.904,E2 4326.904} C_VEL
LIN {X 0,Y 463.844,Z 720.896,A -85,B 0,C 180,E1 4326.126,E2 4326.126} C_VEL
LIN {X 0,Y 463.023,Z 718.823,A -85,B 0,C 180,E1 4324.707,E2 4324.707} C_VEL
LIN {X 0,Y 461.984,Z 714.917,A -85,B 0,C 180,E1 4320.372,E2 4320.372} C_VEL
LIN {X 0,Y 461.986,Z 715.209,A -85,B 0,C 180,E1 4319.256,E2 4319.256} C_VEL
LIN {X 0,Y 463.387,Z 719.663,A -85,B 0,C 180,E1 4314.738,E2 4314.738} C_VEL
LIN {X 0,Y 463.855,Z 721.277,A -85,B 0,C 180,E1 4313.916,E2 4313.916} C_VEL
LIN {X 0,Y 443.969,Z 899.662,A -85,B 0,C 180,E1 4311.497,E2 4311.497} C_VEL
LIN {X 0,Y 439.738,Z 925.722,A -85,B 0,C 180,E1 4311.107,E2 4311.107} C_VEL
LIN {X 0,Y 433.374,Z 953.422,A -85,B 0,C 180,E1 4310.629,E2 4310.629} C_VEL
LIN {X 0,Y 427.195,Z 975.141,A -85,B 0,C 180,E1 4310.155,E2 4310.155} C_VEL
LIN {X 0,Y 420.307,Z 995.792,A -85,B 0,C 180,E1 4309.602,E2 4309.602} C_VEL
LIN {X 0,Y 412.099,Z 1017.175,A -85,B 0,C 180,E1 4308.912,E2 4308.912} C_VEL
LIN {X 0,Y 400.361,Z 1043.609,A -85,B 0,C 180,E1 4307.861,E2 4307.861} C_VEL
LIN {X 0,Y 389.652,Z 1064.573,A -85,B 0,C 180,E1 4306.834,E2 4306.834} C_VEL
LIN {X 0,Y 379.096,Z 1083.276,A -85,B 0,C 180,E1 4305.738,E2 4305.738} C_VEL
LIN {X 0,Y 368.237,Z 1100.816,A -85,B 0,C 180,E1 4304.541,E2 4304.541} C_VEL
LIN {X 0,Y 355.873,Z 1119.168,A -85,B 0,C 180,E1 4303.052,E2 4303.052} C_VEL
LIN {X 0,Y 339.659,Z 1141.076,A -85,B 0,C 180,E1 4300.879,E2 4300.879} C_VEL
LIN {X 0,Y 325.163,Z 1158.853,A -85,B 0,C 180,E1 4298.686,E2 4298.686} C_VEL
LIN {X 0,Y 311.95,Z 1173.984,A -85,B 0,C 180,E1 4296.43,E2 4296.43} C_VEL
LIN {X 0,Y 299.247,Z 1187.671,A -85,B 0,C 180,E1 4293.986,E2 4293.986} C_VEL
LIN {X 0,Y 283.673,Z 1203.581,A -85,B 0,C 180,E1 4290.515,E2 4290.515} C_VEL
LIN {X 0,Y 268.549,Z 1217.95,A -85,B 0,C 180,E1 4286.498,E2 4286.498} C_VEL
LIN {X 0,Y 256.514,Z 1229.011,A -85,B 0,C 180,E1 4282.659,E2 4282.659} C_VEL
LIN {X 0,Y 245.427,Z 1239.01,A -85,B 0,C 180,E1 4278.388,E2 4278.388} C_VEL
LIN {X 0,Y 234.327,Z 1249.043,A -85,B 0,C 180,E1 4273.045,E2 4273.045} C_VEL
LIN {X 0,Y 223.968,Z 1258.533,A -85,B 0,C 180,E1 4266.414,E2 4266.414} C_VEL
LIN {X 0,Y 217.512,Z 1264.871,A -85,B 0,C 180,E1 4260.671,E2 4260.671} C_VEL
LIN {X 0,Y 213.024,Z 1269.81,A -85,B 0,C 180,E1 4254.979,E2 4254.979} C_VEL
LIN {X 0,Y 210.106,Z 1273.688,A -85,B 0,C 180,E1 4249.161,E2 4249.161} C_VEL
LIN {X 0,Y 208.52,Z 1276.552,A -85,B 0,C 180,E1 4243.238,E2 4243.238} C_VEL
LIN {X 0,Y 207.984,Z 1278.276,A -85,B 0,C 180,E1 4237.728,E2 4237.728} C_VEL
LIN {X 0,Y 207.914,Z 1279.032,A -85,B 0,C 180,E1 4233.024,E2 4233.024} C_VEL
LIN {X 0,Y 207.909,Z 1279.143,A -85,B 0,C 180,E1 4228.339,E2 4228.339} C_VEL
LIN {X 0,Y 207.968,Z 1278.471,A -85,B 0,C 180,E1 4223.089,E2 4223.089} C_VEL
LIN {X 0,Y 208.441,Z 1276.736,A -85,B 0,C 180,E1 4217.245,E2 4217.245} C_VEL
LIN {X 0,Y 209.898,Z 1273.98,A -85,B 0,C 180,E1 4211.38,E2 4211.38} C_VEL
LIN {X 0,Y 212.698,Z 1270.188,A -85,B 0,C 180,E1 4205.556,E2 4205.556} C_VEL
LIN {X 0,Y 217.03,Z 1265.335,A -85,B 0,C 180,E1 4199.849,E2 4199.849} C_VEL
LIN {X 0,Y 223.202,Z 1259.197,A -85,B 0,C 180,E1 4194.178,E2 4194.178} C_VEL
LIN {X 0,Y 233.063,Z 1250.167,A -85,B 0,C 180,E1 4187.65,E2 4187.65} C_VEL
LIN {X 0,Y 244.663,Z 1239.633,A -85,B 0,C 180,E1 4181.937,E2 4181.937} C_VEL
LIN {X 0,Y 255.395,Z 1229.94,A -85,B 0,C 180,E1 4177.729,E2 4177.729} C_VEL
LIN {X 0,Y 266.696,Z 1219.556,A -85,B 0,C 180,E1 4174.041,E2 4174.041} C_VEL
LIN {X 0,Y 279.617,Z 1207.293,A -85,B 0,C 180,E1 4170.474,E2 4170.474} C_VEL
LIN {X 0,Y 296.368,Z 1190.582,A -85,B 0,C 180,E1 4166.605,E2 4166.605} C_VEL
LIN {X 0,Y 311.218,Z 1174.624,A -85,B 0,C 180,E1 4163.694,E2 4163.694} C_VEL
LIN {X 0,Y 324.007,Z 1160.015,A -85,B 0,C 180,E1 4161.491,E2 4161.491} C_VEL
LIN {X 0,Y 336.844,Z 1144.36,A -85,B 0,C 180,E1 4159.514,E2 4159.514} C_VEL
LIN {X 0,Y 352.128,Z 1124.291,A -85,B 0,C 180,E1 4157.422,E2 4157.422} C_VEL
LIN {X 0,Y 367.091,Z 1102.293,A -85,B 0,C 180,E1 4155.584,E2 4155.584} C_VEL
LIN {X 0,Y 378.411,Z 1084.081,A -85,B 0,C 180,E1 4154.325,E2 4154.325} C_VEL
LIN {X 0,Y 388.936,Z 1065.504,A -85,B 0,C 180,E1 4153.227,E2 4153.227} C_VEL
LIN {X 0,Y 399.501,Z 1044.915,A -85,B 0,C 180,E1 4152.208,E2 4152.208} C_VEL
LIN {X 0,Y 411.231,Z 1018.805,A -85,B 0,C 180,E1 4151.153,E2 4151.153} C_VEL
LIN {X 0,Y 419.889,Z 996.344,A -85,B 0,C 180,E1 4150.421,E2 4150.421} C_VEL
LIN {X 0,Y 426.821,Z 975.624,A -85,B 0,C 180,E1 4149.864,E2 4149.864} C_VEL
LIN {X 0,Y 433.038,Z 953.833,A -85,B 0,C 180,E1 4149.385,E2 4149.385} C_VEL
LIN {X 0,Y 439.376,Z 926.471,A -85,B 0,C 180,E1 4148.909,E2 4148.909} C_VEL
LIN {X 0,Y 443.702,Z 899.923,A -85,B 0,C 180,E1 4148.512,E2 4148.512} C_VEL
LIN {X 0,Y 460.219,Z 751.702,A -85,B 0,C 180,E1 4146.497,E2 4146.497} C_VEL
LIN {X 0,Y 463.653,Z 720.759,A -85,B 0,C 180,E1 4146.066,E2 4146.066} C_VEL
LIN {X 0,Y 462.851,Z 718.715,A -85,B 0,C 180,E1 4144.709,E2 4144.709} C_VEL
LIN {X 0,Y 461.735,Z 714.839,A -85,B 0,C 180,E1 4140.62,E2 4140.62} C_VEL
LIN {X 0,Y 461.748,Z 715.03,A -85,B 0,C 180,E1 4138.883,E2 4138.883} C_VEL
LIN {X 0,Y 463.228,Z 719.591,A -85,B 0,C 180,E1 4134.426,E2 4134.426} C_VEL
LIN {X 0,Y 463.624,Z 720.854,A -85,B 0,C 180,E1 4133.755,E2 4133.755} C_VEL
LIN {X 0,Y 443.849,Z 898.208,A -85,B 0,C 180,E1 4131.351,E2 4131.351} C_VEL
LIN {X 0,Y 439.634,Z 924.151,A -85,B 0,C 180,E1 4130.964,E2 4130.964} C_VEL
LIN {X 0,Y 433.322,Z 951.738,A -85,B 0,C 180,E1 4130.47,E2 4130.47} C_VEL
LIN {X 0,Y 427.23,Z 973.248,A -85,B 0,C 180,E1 4129.979,E2 4129.979} C_VEL
LIN {X 0,Y 420.602,Z 993.229,A -85,B 0,C 180,E1 4129.429,E2 4129.429} C_VEL
LIN {X 0,Y 412.881,Z 1013.522,A -85,B 0,C 180,E1 4128.762,E2 4128.762} C_VEL
LIN {X 0,Y 402.983,Z 1036.392,A -85,B 0,C 180,E1 4127.857,E2 4127.857} C_VEL
LIN {X 0,Y 390.524,Z 1061.239,A -85,B 0,C 180,E1 4126.648,E2 4126.648} C_VEL
LIN {X 0,Y 379.707,Z 1080.457,A -85,B 0,C 180,E1 4125.513,E2 4125.513} C_VEL
LIN {X 0,Y 368.761,Z 1098.18,A -85,B 0,C 180,E1 4124.282,E2 4124.282} C_VEL
LIN {X 0,Y 356.858,Z 1115.849,A -85,B 0,C 180,E1 4122.841,E2 4122.841} C_VEL
LIN {X 0,Y 341.515,Z 1136.76,A -85,B 0,C 180,E1 4120.779,E2 4120.779} C_VEL
LIN {X 0,Y 325.837,Z 1155.93,A -85,B 0,C 180,E1 4118.412,E2 4118.412} C_VEL
LIN {X 0,Y 312.662,Z 1170.945,A -85,B 0,C 180,E1 4116.159,E2 4116.159} C_VEL
LIN {X 0,Y 299.269,Z 1185.282,A -85,B 0,C 180,E1 4113.569,E2 4113.569} C_VEL
LIN {X 0,Y 282.833,Z 1201.818,A -85,B 0,C 180,E1 4109.867,E2 4109.867} C_VEL
LIN {X 0,Y 268.104,Z 1215.638,A -85,B 0,C 180,E1 4105.895,E2 4105.895} C_VEL
LIN {X 0,Y 256.746,Z 1225.933,A -85,B 0,C 180,E1 4102.246,E2 4102.246} C_VEL
LIN {X 0,Y 245.94,Z 1235.529,A -85,B 0,C 180,E1 4098.08,E2 4098.08} C_VEL
LIN {X 0,Y 234.193,Z 1245.946,A -85,B 0,C 180,E1 4092.429,E2 4092.429} C_VEL
LIN {X 0,Y 224.274,Z 1254.774,A -85,B 0,C 180,E1 4086.058,E2 4086.058} C_VEL
LIN {X 0,Y 217.792,Z 1260.94,A -85,B 0,C 180,E1 4080.332,E2 4080.332} C_VEL
LIN {X 0,Y 213.271,Z 1265.712,A -85,B 0,C 180,E1 4074.669,E2 4074.669} C_VEL
LIN {X 0,Y 210.276,Z 1269.446,A -85,B 0,C 180,E1 4068.866,E2 4068.866} C_VEL
LIN {X 0,Y 208.649,Z 1272.156,A -85,B 0,C 180,E1 4063.024,E2 4063.024} C_VEL
LIN {X 0,Y 208.022,Z 1273.941,A -85,B 0,C 180,E1 4056.909,E2 4056.909} C_VEL
LIN {X 0,Y 207.905,Z 1274.615,A -85,B 0,C 180,E1 4051.386,E2 4051.386} C_VEL
LIN {X 0,Y 207.938,Z 1274.404,A -85,B 0,C 180,E1 4045.872,E2 4045.872} C_VEL
LIN {X 0,Y 208.182,Z 1273.31,A -85,B 0,C 180,E1 4040.331,E2 4040.331} C_VEL
LIN {X 0,Y 209.483,Z 1270.765,A -85,B 0,C 180,E1 4033.367,E2 4033.367} C_VEL
LIN {X 0,Y 212.693,Z 1266.427,A -85,B 0,C 180,E1 4026.163,E2 4026.163} C_VEL
LIN {X 0,Y 217.221,Z 1261.562,A -85,B 0,C 180,E1 4020.2,E2 4020.2} C_VEL
LIN {X 0,Y 223.501,Z 1255.523,A -85,B 0,C 180,E1 4014.449,E2 4014.449} C_VEL
LIN {X 0,Y 231.559,Z 1248.264,A -85,B 0,C 180,E1 4008.99,E2 4008.99} C_VEL
LIN {X 0,Y 243.774,Z 1237.565,A -85,B 0,C 180,E1 4002.773,E2 4002.773} C_VEL
LIN {X 0,Y 256.014,Z 1226.679,A -85,B 0,C 180,E1 3997.928,E2 3997.928} C_VEL
LIN {X 0,Y 267.932,Z 1215.899,A -85,B 0,C 180,E1 3994.072,E2 3994.072} C_VEL
LIN {X 0,Y 280.882,Z 1203.761,A -85,B 0,C 180,E1 3990.533,E2 3990.533} C_VEL
LIN {X 0,Y 298.362,Z 1186.397,A -85,B 0,C 180,E1 3986.537,E2 3986.537} C_VEL
LIN {X 0,Y 311.72,Z 1172.164,A -85,B 0,C 180,E1 3983.93,E2 3983.93} C_VEL
LIN {X 0,Y 324.87,Z 1157.26,A -85,B 0,C 180,E1 3981.664,E2 3981.664} C_VEL
LIN {X 0,Y 338.147,Z 1141.149,A -85,B 0,C 180,E1 3979.623,E2 3979.623} C_VEL
LIN {X 0,Y 353.761,Z 1120.619,A -85,B 0,C 180,E1 3977.484,E2 3977.484} C_VEL
LIN {X 0,Y 367.738,Z 1100.088,A -85,B 0,C 180,E1 3975.76,E2 3975.76} C_VEL
LIN {X 0,Y 378.962,Z 1082.06,A -85,B 0,C 180,E1 3974.487,E2 3974.487} C_VEL
LIN {X 0,Y 389.48,Z 1063.541,A -85,B 0,C 180,E1 3973.379,E2 3973.379} C_VEL
LIN {X 0,Y 400.139,Z 1042.772,A -85,B 0,C 180,E1 3972.33,E2 3972.33} C_VEL
LIN {X 0,Y 411.827,Z 1016.7,A -85,B 0,C 180,E1 3971.255,E2 3971.255} C_VEL
LIN {X 0,Y 419.997,Z 995.558,A -85,B 0,C 180,E1 3970.544,E2 3970.544} C_VEL
LIN {X 0,Y 427.017,Z 974.664,A -85,B 0,C 180,E1 3969.961,E2 3969.961} C_VEL
LIN {X 0,Y 433.018,Z 953.733,A -85,B 0,C 180,E1 3969.476,E2 3969.476} C_VEL
LIN {X 0,Y 438.502,Z 930.641,A -85,B 0,C 180,E1 3969.045,E2 3969.045} C_VEL
LIN {X 0,Y 443.753,Z 900.715,A -85,B 0,C 180,E1 3968.589,E2 3968.589} C_VEL
LIN {X 0,Y 451,Z 837.113,A -85,B 0,C 180,E1 3967.717,E2 3967.717} C_VEL
LIN {X 0,Y 457.629,Z 776.927,A -85,B 0,C 180,E1 3966.904,E2 3966.904} C_VEL
LIN {X 0,Y 458.344,Z 769.409,A -85,B 0,C 180,E1 3966.676,E2 3966.676} C_VEL
LIN {X 0,Y 459.861,Z 749.916,A -85,B 0,C 180,E1 3965.637,E2 3965.637} C_VEL
LIN {X 0,Y 460.523,Z 743.446,A -85,B 0,C 180,E1 3965.461,E2 3965.461} C_VEL
LIN {X 0,Y 462.323,Z 727.525,A -85,B 0,C 180,E1 3965.243,E2 3965.243} C_VEL
LIN {X 0,Y 461.009,Z 722.857,A -85,B 0,C 180,E1 3960.373,E2 3960.373} C_VEL
LIN {X 0,Y 461.005,Z 723.088,A -85,B 0,C 180,E1 3959.379,E2 3959.379} C_VEL
LIN {X 0,Y 462.343,Z 727.619,A -85,B 0,C 180,E1 3954.824,E2 3954.824} C_VEL
LIN {X 0,Y 442.852,Z 899.595,A -85,B 0,C 180,E1 3952.525,E2 3952.525} C_VEL
LIN {X 0,Y 438.556,Z 925.713,A -85,B 0,C 180,E1 3952.144,E2 3952.144} C_VEL
LIN {X 0,Y 432.137,Z 953.345,A -85,B 0,C 180,E1 3951.682,E2 3951.682} C_VEL
LIN {X 0,Y 425.859,Z 975.163,A -85,B 0,C 180,E1 3951.221,E2 3951.221} C_VEL
LIN {X 0,Y 418.786,Z 996.093,A -85,B 0,C 180,E1 3950.679,E2 3950.679} C_VEL
LIN {X 0,Y 410.158,Z 1018.225,A -85,B 0,C 180,E1 3949.984,E2 3949.984} C_VEL
LIN {X 0,Y 397.818,Z 1045.33,A -85,B 0,C 180,E1 3948.925,E2 3948.925} C_VEL
LIN {X 0,Y 387.424,Z 1065.302,A -85,B 0,C 180,E1 3947.967,E2 3947.967} C_VEL
LIN {X 0,Y 376.717,Z 1083.927,A -85,B 0,C 180,E1 3946.9,E2 3946.9} C_VEL
LIN {X 0,Y 365.256,Z 1102.069,A -85,B 0,C 180,E1 3945.685,E2 3945.685} C_VEL
LIN {X 0,Y 350.244,Z 1123.791,A -85,B 0,C 180,E1 3943.923,E2 3943.923} C_VEL
LIN {X 0,Y 334.53,Z 1144.04,A -85,B 0,C 180,E1 3941.869,E2 3941.869} C_VEL
LIN {X 0,Y 321.423,Z 1159.695,A -85,B 0,C 180,E1 3939.94,E2 3939.94} C_VEL
LIN {X 0,Y 307.926,Z 1174.745,A -85,B 0,C 180,E1 3937.715,E2 3937.715} C_VEL
LIN {X 0,Y 292.684,Z 1190.679,A -85,B 0,C 180,E1 3934.846,E2 3934.846} C_VEL
LIN {X 0,Y 276.12,Z 1206.71,A -85,B 0,C 180,E1 3931.186,E2 3931.186} C_VEL
LIN {X 0,Y 262.699,Z 1219.014,A -85,B 0,C 180,E1 3927.654,E2 3927.654} C_VEL
LIN {X 0,Y 250.307,Z 1229.958,A -85,B 0,C 180,E1 3923.781,E2 3923.781} C_VEL
LIN {X 0,Y 237.824,Z 1240.758,A -85,B 0,C 180,E1 3919.014,E2 3919.014} C_VEL
LIN {X 0,Y 224.712,Z 1251.94,A -85,B 0,C 180,E1 3912.546,E2 3912.546} C_VEL
LIN {X 0,Y 216.232,Z 1259.362,A -85,B 0,C 180,E1 3906.94,E2 3906.94} C_VEL
LIN {X 0,Y 209.848,Z 1265.296,A -85,B 0,C 180,E1 3901.279,E2 3901.279} C_VEL
LIN {X 0,Y 205.169,Z 1270.139,A -85,B 0,C 180,E1 3895.386,E2 3895.386} C_VEL
LIN {X 0,Y 202.009,Z 1274.106,A -85,B 0,C 180,E1 3889.02,E2 3889.02} C_VEL
LIN {X 0,Y 200.301,Z 1277.248,A -85,B 0,C 180,E1 3881.801,E2 3881.801} C_VEL
LIN {X 0,Y 199.926,Z 1278.78,A -85,B 0,C 180,E1 3875.156,E2 3875.156} C_VEL
LIN {X 0,Y 199.893,Z 1279.17,A -85,B 0,C 180,E1 3869.705,E2 3869.705} C_VEL
LIN {X 0,Y 199.942,Z 1278.659,A -85,B 0,C 180,E1 3863.964,E2 3863.964} C_VEL
LIN {X 0,Y 200.424,Z 1276.878,A -85,B 0,C 180,E1 3857.312,E2 3857.312} C_VEL
LIN {X 0,Y 202.139,Z 1273.89,A -85,B 0,C 180,E1 3850.637,E2 3850.637} C_VEL
LIN {X 0,Y 205.176,Z 1270.097,A -85,B 0,C 180,E1 3844.598,E2 3844.598} C_VEL
LIN {X 0,Y 209.862,Z 1265.243,A -85,B 0,C 180,E1 3838.705,E2 3838.705} C_VEL
LIN {X 0,Y 216.248,Z 1259.296,A -85,B 0,C 180,E1 3833.044,E2 3833.044} C_VEL
LIN {X 0,Y 225.431,Z 1251.283,A -85,B 0,C 180,E1 3827.042,E2 3827.042} C_VEL
LIN {X 0,Y 238.586,Z 1240.002,A -85,B 0,C 180,E1 3820.656,E2 3820.656} C_VEL
LIN {X 0,Y 250.333,Z 1229.847,A -85,B 0,C 180,E1 3816.205,E2 3816.205} C_VEL
LIN {X 0,Y 262.08,Z 1219.462,A -85,B 0,C 180,E1 3812.517,E2 3812.517} C_VEL
LIN {X 0,Y 275.453,Z 1207.199,A -85,B 0,C 180,E1 3808.968,E2 3808.968} C_VEL
LIN {X 0,Y 292.715,Z 1190.488,A -85,B 0,C 180,E1 3805.14,E2 3805.14} C_VEL
LIN {X 0,Y 307.959,Z 1174.53,A -85,B 0,C 180,E1 3802.272,E2 3802.272} C_VEL
LIN {X 0,Y 321.052,Z 1159.921,A -85,B 0,C 180,E1 3800.109,E2 3800.109} C_VEL
LIN {X 0,Y 334.149,Z 1144.283,A -85,B 0,C 180,E1 3798.175,E2 3798.175} C_VEL
LIN {X 0,Y 349.742,Z 1124.197,A -85,B 0,C 180,E1 3796.129,E2 3796.129} C_VEL
LIN {X 0,Y 364.857,Z 1102.365,A -85,B 0,C 180,E1 3794.35,E2 3794.35} C_VEL
LIN {X 0,Y 376.31,Z 1084.245,A -85,B 0,C 180,E1 3793.131,E2 3793.131} C_VEL
LIN {X 0,Y 387.012,Z 1065.653,A -85,B 0,C 180,E1 3792.062,E2 3792.062} C_VEL
LIN {X 0,Y 397.858,Z 1044.82,A -85,B 0,C 180,E1 3791.061,E2 3791.061} C_VEL
LIN {X 0,Y 409.739,Z 1018.71,A -85,B 0,C 180,E1 3790.04,E2 3790.04} C_VEL
LIN {X 0,Y 418.501,Z 996.248,A -85,B 0,C 180,E1 3789.332,E2 3789.332} C_VEL
LIN {X 0,Y 425.467,Z 975.673,A -85,B 0,C 180,E1 3788.797,E2 3788.797} C_VEL
